LIN {X 0,Y 418.326,Z 381.944,A -85,B 0,C 180,E1 -10142.828,E2 -10142.828} C_VEL
LIN {X 0,Y 420.764,Z 394.079,A -85,B 0,C 180,E1 -10145.581,E2 -10145.581} C_VEL
LIN {X 0,Y 421.234,Z 397.819,A -85,B 0,C 180,E1 -10146.395,E2 -10146.395} C_VEL
LIN {X 0,Y 420.167,Z 413.645,A -85,B 0,C 180,E1 -10149.637,E2 -10149.637} C_VEL
LIN {X 0,Y 419.768,Z 420.199,A -85,B 0,C 180,E1 -10150.945,E2 -10150.945} C_VEL
LIN {X 0,Y 423.831,Z 444.894,A -85,B 0,C 180,E1 -10151.565,E2 -10151.565} C_VEL
LIN {X 0,Y 422.879,Z 528.082,A -85,B 0,C 180,E1 -10152.998,E2 -10152.998} C_VEL
LIN {X 0,Y 422.43,Z 541.332,A -85,B 0,C 180,E1 -10153.415,E2 -10153.415} C_VEL
LIN {X 0,Y 421.773,Z 553.48,A -85,B 0,C 180,E1 -10153.979,E2 -10153.979} C_VEL
LIN {X 0,Y 421.045,Z 565.74,A -85,B 0,C 180,E1 -10154.758,E2 -10154.758} C_VEL
LIN {X 0,Y 420.246,Z 576.923,A -85,B 0,C 180,E1 -10155.68,E2 -10155.68} C_VEL
LIN {X 0,Y 419.549,Z 587.766,A -85,B 0,C 180,E1 -10156.806,E2 -10156.806} C_VEL
LIN {X 0,Y 418.988,Z 596.3,A -85,B 0,C 180,E1 -10157.897,E2 -10157.897} C_VEL
LIN {X 0,Y 418.329,Z 604.171,A -85,B 0,C 180,E1 -10159.105,E2 -10159.105} C_VEL
LIN {X 0,Y 417.793,Z 611.86,A -85,B 0,C 180,E1 -10160.56,E2 -10160.56} C_VEL
LIN {X 0,Y 417.393,Z 618.951,A -85,B 0,C 180,E1 -10162.258,E2 -10162.258} C_VEL
LIN {X 0,Y 417.15,Z 623.713,A -85,B 0,C 180,E1 -10163.728,E2 -10163.728} C_VEL
LIN {X 0,Y 417.114,Z 627.274,A -85,B 0,C 180,E1 -10165.167,E2 -10165.167} C_VEL
LIN {X 0,Y 417,Z 629.132,A -85,B 0,C 180,E1 -10166.134,E2 -10166.134} C_VEL
LIN {X 0,Y 417.018,Z 630.527,A -85,B 0,C 180,E1 -10167.102,E2 -10167.102} C_VEL
LIN {X 0,Y 417.055,Z 631.523,A -85,B 0,C 180,E1 -10168.068,E2 -10168.068} C_VEL
LIN {X 0,Y 416.982,Z 632.345,A -85,B 0,C 180,E1 -10170,E2 -10170} C_VEL
LIN {X 0,Y 417.055,Z 631.522,A -85,B 0,C 180,E1 -10171.931,E2 -10171.931} C_VEL
LIN {X 0,Y 417.018,Z 630.526,A -85,B 0,C 180,E1 -10172.898,E2 -10172.898} C_VEL
LIN {X 0,Y 417,Z 629.129,A -85,B 0,C 180,E1 -10173.865,E2 -10173.865} C_VEL
LIN {X 0,Y 417.137,Z 626.196,A -85,B 0,C 180,E1 -10175.317,E2 -10175.317} C_VEL
LIN {X 0,Y 417.235,Z 622.223,A -85,B 0,C 180,E1 -10176.771,E2 -10176.771} C_VEL
LIN {X 0,Y 417.542,Z 616.116,A -85,B 0,C 180,E1 -10178.469,E2 -10178.469} C_VEL
LIN {X 0,Y 417.955,Z 609.442,A -85,B 0,C 180,E1 -10179.925,E2 -10179.925} C_VEL
LIN {X 0,Y 418.541,Z 601.164,A -85,B 0,C 180,E1 -10181.379,E2 -10181.379} C_VEL
LIN {X 0,Y 419.25,Z 592.68,A -85,B 0,C 180,E1 -10182.587,E2 -10182.587} C_VEL
LIN {X 0,Y 419.898,Z 582.125,A -85,B 0,C 180,E1 -10183.805,E2 -10183.805} C_VEL
LIN {X 0,Y 420.714,Z 570.388,A -85,B 0,C 180,E1 -10184.882,E2 -10184.882} C_VEL
LIN {X 0,Y 421.47,Z 558.517,A -85,B 0,C 180,E1 -10185.722,E2 -10185.722} C_VEL
LIN {X 0,Y 422.196,Z 546.166,A -85,B 0,C 180,E1 -10186.376,E2 -10186.376} C_VEL
LIN {X 0,Y 422.663,Z 533.478,A -85,B 0,C 180,E1 -10186.855,E2 -10186.855} C_VEL
LIN {X 0,Y 423.062,Z 520.188,A -85,B 0,C 180,E1 -10187.149,E2 -10187.149} C_VEL
LIN {X 0,Y 423.713,Z 444.119,A -85,B 0,C 180,E1 -10188.448,E2 -10188.448} C_VEL
LIN {X 0,Y 419.753,Z 419.907,A -85,B 0,C 180,E1 -10189.078,E2 -10189.078} C_VEL
LIN {X 0,Y 421.027,Z 401.735,A -85,B 0,C 180,E1 -10192.787,E2 -10192.787} C_VEL
LIN {X 0,Y 421.181,Z 396.537,A -85,B 0,C 180,E1 -10193.869,E2 -10193.869} C_VEL
LIN {X 0,Y 419.001,Z 385.302,A -85,B 0,C 180,E1 -10196.391,E2 -10196.391} C_VEL
LIN {X 0,Y 418.336,Z 381.878,A -85,B 0,C 180,E1 -10197.208,E2 -10197.208} C_VEL
LIN {X 0,Y 418.247,Z 381.882,A -85,B 0,C 180,E1 -10200.272,E2 -10200.272} C_VEL
LIN {X 0,Y 418.25,Z 381.883,A -85,B 0,C 180,E1 -10203.677,E2 -10203.677} C_VEL
LIN {X 0,Y 418.242,Z 381.888,A -85,B 0,C 180,E1 -10207.224,E2 -10207.224} C_VEL
LIN {X 0,Y 418.253,Z 381.882,A -85,B 0,C 180,E1 -10209.682,E2 -10209.682} C_VEL
LIN {X 0,Y 418.231,Z 381.885,A -85,B 0,C 180,E1 -10212.321,E2 -10212.321} C_VEL
LIN {X 0,Y 418.241,Z 381.888,A -85,B 0,C 180,E1 -10215.109,E2 -10215.109} C_VEL
LIN {X 0,Y 418.244,Z 381.883,A -85,B 0,C 180,E1 -10217.767,E2 -10217.767} C_VEL
LIN {X 0,Y 418.257,Z 381.886,A -85,B 0,C 180,E1 -10220.619,E2 -10220.619} C_VEL
LIN {X 0,Y 418.245,Z 381.883,A -85,B 0,C 180,E1 -10223.976,E2 -10223.976} C_VEL
LIN {X 0,Y 418.259,Z 381.883,A -85,B 0,C 180,E1 -10227.156,E2 -10227.156} C_VEL
LIN {X 0,Y 418.27,Z 381.884,A -85,B 0,C 180,E1 -10230.895,E2 -10230.895} C_VEL
LIN {X 0,Y 418.271,Z 381.881,A -85,B 0,C 180,E1 -10234.096,E2 -10234.096} C_VEL
LIN {X 0,Y 418.24,Z 381.884,A -85,B 0,C 180,E1 -10237.264,E2 -10237.264} C_VEL
LIN {X 0,Y 418.286,Z 381.883,A -85,B 0,C 180,E1 -10240.364,E2 -10240.364} C_VEL
LIN {X 0,Y 418.32,Z 381.873,A -85,B 0,C 180,E1 -10243.405,E2 -10243.405} C_VEL
LIN {X 0,Y 418.358,Z 381.87,A -85,B 0,C 180,E1 -10246.994,E2 -10246.994} C_VEL
LIN {X 0,Y 418.36,Z 381.875,A -85,B 0,C 180,E1 -10250.329,E2 -10250.329} C_VEL
LIN {X 0,Y 418.48,Z 381.853,A -85,B 0,C 180,E1 -10253.249,E2 -10253.249} C_VEL
LIN {X 0,Y 418.341,Z 381.871,A -85,B 0,C 180,E1 -10255.182,E2 -10255.182} C_VEL
LIN {X 0,Y 418.545,Z 381.85,A -85,B 0,C 180,E1 -10258.076,E2 -10258.076} C_VEL
LIN {X 0,Y 418.674,Z 381.834,A -85,B 0,C 180,E1 -10260,E2 -10260} C_VEL
LIN {X 0,Y 418.513,Z 381.85,A -85,B 0,C 180,E1 -10262.888,E2 -10262.888} C_VEL
LIN {X 0,Y 418.497,Z 381.852,A -85,B 0,C 180,E1 -10266.751,E2 -10266.751} C_VEL
LIN {X 0,Y 418.403,Z 381.864,A -85,B 0,C 180,E1 -10268.695,E2 -10268.695} C_VEL
LIN {X 0,Y 418.358,Z 381.87,A -85,B 0,C 180,E1 -10272.614,E2 -10272.614} C_VEL
LIN {X 0,Y 418.305,Z 381.878,A -85,B 0,C 180,E1 -10275.594,E2 -10275.594} C_VEL
LIN {X 0,Y 418.288,Z 381.878,A -85,B 0,C 180,E1 -10278.617,E2 -10278.617} C_VEL
LIN {X 0,Y 418.237,Z 381.888,A -85,B 0,C 180,E1 -10281.696,E2 -10281.696} C_VEL
LIN {X 0,Y 418.286,Z 381.877,A -85,B 0,C 180,E1 -10284.865,E2 -10284.865} C_VEL
LIN {X 0,Y 418.296,Z 381.88,A -85,B 0,C 180,E1 -10288.063,E2 -10288.063} C_VEL
LIN {X 0,Y 418.218,Z 381.889,A -85,B 0,C 180,E1 -10291.396,E2 -10291.396} C_VEL
LIN {X 0,Y 418.268,Z 381.88,A -85,B 0,C 180,E1 -10294.58,E2 -10294.58} C_VEL
LIN {X 0,Y 418.237,Z 381.888,A -85,B 0,C 180,E1 -10297.835,E2 -10297.835} C_VEL
LIN {X 0,Y 418.263,Z 381.881,A -85,B 0,C 180,E1 -10300.943,E2 -10300.943} C_VEL
LIN {X 0,Y 418.219,Z 381.891,A -85,B 0,C 180,E1 -10303.731,E2 -10303.731} C_VEL
LIN {X 0,Y 418.211,Z 381.887,A -85,B 0,C 180,E1 -10306.449,E2 -10306.449} C_VEL
LIN {X 0,Y 418.225,Z 381.888,A -85,B 0,C 180,E1 -10309.13,E2 -10309.13} C_VEL
LIN {X 0,Y 418.236,Z 381.884,A -85,B 0,C 180,E1 -10312.166,E2 -10312.166} C_VEL
LIN {X 0,Y 418.268,Z 381.886,A -85,B 0,C 180,E1 -10315.42,E2 -10315.42} C_VEL
LIN {X 0,Y 418.214,Z 381.887,A -85,B 0,C 180,E1 -10318.604,E2 -10318.604} C_VEL
LIN {X 0,Y 418.294,Z 381.877,A -85,B 0,C 180,E1 -10321.937,E2 -10321.937} C_VEL
LIN {X 0,Y 418.304,Z 381.881,A -85,B 0,C 180,E1 -10325.693,E2 -10325.693} C_VEL
LIN {X 0,Y 418.303,Z 381.998,A -85,B 0,C 180,E1 -10326.121,E2 -10326.121} C_VEL
LIN {X 0,Y 420.404,Z 393.102,A -85,B 0,C 180,E1 -10328.936,E2 -10328.936} C_VEL
LIN {X 0,Y 420.115,Z 399.607,A -85,B 0,C 180,E1 -10330.453,E2 -10330.453} C_VEL
LIN {X 0,Y 419.951,Z 402.004,A -85,B 0,C 180,E1 -10331.004,E2 -10331.004} C_VEL
LIN {X 0,Y 424.021,Z 422.399,A -85,B 0,C 180,E1 -10331.562,E2 -10331.562} C_VEL
LIN {X 0,Y 423.027,Z 509.467,A -85,B 0,C 180,E1 -10333.067,E2 -10333.067} C_VEL
LIN {X 0,Y 422.58,Z 522.544,A -85,B 0,C 180,E1 -10333.484,E2 -10333.484} C_VEL
LIN {X 0,Y 422.003,Z 535.695,A -85,B 0,C 180,E1 -10334.113,E2 -10334.113} C_VEL
LIN {X 0,Y 421.338,Z 547.544,A -85,B 0,C 180,E1 -10334.893,E2 -10334.893} C_VEL
LIN {X 0,Y 420.71,Z 558.93,A -85,B 0,C 180,E1 -10335.861,E2 -10335.861} C_VEL
LIN {X 0,Y 420,Z 569.148,A -85,B 0,C 180,E1 -10336.944,E2 -10336.944} C_VEL
LIN {X 0,Y 419.248,Z 578.338,A -85,B 0,C 180,E1 -10338.15,E2 -10338.15} C_VEL
LIN {X 0,Y 418.538,Z 587.261,A -85,B 0,C 180,E1 -10339.601,E2 -10339.601} C_VEL
LIN {X 0,Y 418.021,Z 594.443,A -85,B 0,C 180,E1 -10341.053,E2 -10341.053} C_VEL
LIN {X 0,Y 417.861,Z 596.308,A -85,B 0,C 180,E1 -10341.496,E2 -10341.496} C_VEL
LIN {X 0,Y 416.976,Z 599.134,A -85,B 0,C 180,E1 -10342.2,E2 -10342.2} C_VEL
LIN {X 0,Y 412.546,Z 604.702,A -85,B 0,C 180,E1 -10343.85,E2 -10343.85} C_VEL
LIN {X 0,Y 410.488,Z 607.256,A -85,B 0,C 180,E1 -10344.856,E2 -10344.856} C_VEL
LIN {X 0,Y 410.102,Z 608.331,A -85,B 0,C 180,E1 -10345.384,E2 -10345.384} C_VEL
LIN {X 0,Y 410.033,Z 611.029,A -85,B 0,C 180,E1 -10347.053,E2 -10347.053} C_VEL
LIN {X 0,Y 410.011,Z 612.026,A -85,B 0,C 180,E1 -10348.036,E2 -10348.036} C_VEL
LIN {X 0,Y 409.907,Z 612.876,A -85,B 0,C 180,E1 -10350,E2 -10350} C_VEL
LIN {X 0,Y 409.939,Z 612.687,A -85,B 0,C 180,E1 -10350.983,E2 -10350.983} C_VEL
LIN {X 0,Y 410.011,Z 612.101,A -85,B 0,C 180,E1 -10351.965,E2 -10351.965} C_VEL
LIN {X 0,Y 410.033,Z 611.134,A -85,B 0,C 180,E1 -10352.948,E2 -10352.948} C_VEL
LIN {X 0,Y 410.02,Z 609.779,A -85,B 0,C 180,E1 -10353.932,E2 -10353.932} C_VEL
LIN {X 0,Y 410.258,Z 606.908,A -85,B 0,C 180,E1 -10355.407,E2 -10355.407} C_VEL
LIN {X 0,Y 410.43,Z 603.021,A -85,B 0,C 180,E1 -10356.885,E2 -10356.885} C_VEL
LIN {X 0,Y 410.747,Z 598.003,A -85,B 0,C 180,E1 -10358.363,E2 -10358.363} C_VEL
LIN {X 0,Y 411.233,Z 591.687,A -85,B 0,C 180,E1 -10359.84,E2 -10359.84} C_VEL
LIN {X 0,Y 411.887,Z 583.778,A -85,B 0,C 180,E1 -10361.316,E2 -10361.316} C_VEL
LIN {X 0,Y 412.532,Z 575.717,A -85,B 0,C 180,E1 -10362.546,E2 -10362.546} C_VEL
LIN {X 0,Y 413.313,Z 565.878,A -85,B 0,C 180,E1 -10363.772,E2 -10363.772} C_VEL
LIN {X 0,Y 414.013,Z 554.816,A -85,B 0,C 180,E1 -10364.878,E2 -10364.878} C_VEL
LIN {X 0,Y 414.727,Z 543.966,A -85,B 0,C 180,E1 -10365.732,E2 -10365.732} C_VEL
LIN {X 0,Y 415.441,Z 531.98,A -85,B 0,C 180,E1 -10366.461,E2 -10366.461} C_VEL
LIN {X 0,Y 415.942,Z 518.813,A -85,B 0,C 180,E1 -10367.041,E2 -10367.041} C_VEL
LIN {X 0,Y 416.334,Z 505.543,A -85,B 0,C 180,E1 -10367.404,E2 -10367.404} C_VEL
LIN {X 0,Y 417.21,Z 422.842,A -85,B 0,C 180,E1 -10368.842,E2 -10368.842} C_VEL
LIN {X 0,Y 413.089,Z 402.156,A -85,B 0,C 180,E1 -10369.42,E2 -10369.42} C_VEL
LIN {X 0,Y 413.501,Z 394.743,A -85,B 0,C 180,E1 -10371.173,E2 -10371.173} C_VEL
LIN {X 0,Y 411.268,Z 382.832,A -85,B 0,C 180,E1 -10374.244,E2 -10374.244} C_VEL
LIN {X 0,Y 411.262,Z 382.758,A -85,B 0,C 180,E1 -10377.478,E2 -10377.478} C_VEL
LIN {X 0,Y 411.193,Z 382.768,A -85,B 0,C 180,E1 -10380.848,E2 -10380.848} C_VEL
LIN {X 0,Y 411.209,Z 382.762,A -85,B 0,C 180,E1 -10384.334,E2 -10384.334} C_VEL
LIN {X 0,Y 411.197,Z 382.761,A -85,B 0,C 180,E1 -10387.974,E2 -10387.974} C_VEL
LIN {X 0,Y 411.167,Z 382.765,A -85,B 0,C 180,E1 -10391.228,E2 -10391.228} C_VEL
LIN {X 0,Y 411.181,Z 382.769,A -85,B 0,C 180,E1 -10394.49,E2 -10394.49} C_VEL
LIN {X 0,Y 411.193,Z 382.764,A -85,B 0,C 180,E1 -10398.196,E2 -10398.196} C_VEL
LIN {X 0,Y 411.228,Z 382.76,A -85,B 0,C 180,E1 -10400.777,E2 -10400.777} C_VEL
LIN {X 0,Y 411.203,Z 382.766,A -85,B 0,C 180,E1 -10404.472,E2 -10404.472} C_VEL
LIN {X 0,Y 411.211,Z 382.76,A -85,B 0,C 180,E1 -10406.873,E2 -10406.873} C_VEL
LIN {X 0,Y 411.243,Z 382.758,A -85,B 0,C 180,E1 -10410.643,E2 -10410.643} C_VEL
LIN {X 0,Y 411.242,Z 382.756,A -85,B 0,C 180,E1 -10413.619,E2 -10413.619} C_VEL
LIN {X 0,Y 411.207,Z 382.76,A -85,B 0,C 180,E1 -10416.853,E2 -10416.853} C_VEL
LIN {X 0,Y 411.269,Z 382.757,A -85,B 0,C 180,E1 -10420.031,E2 -10420.031} C_VEL
LIN {X 0,Y 411.268,Z 382.752,A -85,B 0,C 180,E1 -10423.131,E2 -10423.131} C_VEL
LIN {X 0,Y 411.31,Z 382.746,A -85,B 0,C 180,E1 -10426.896,E2 -10426.896} C_VEL
LIN {X 0,Y 411.297,Z 382.753,A -85,B 0,C 180,E1 -10430.161,E2 -10430.161} C_VEL
LIN {X 0,Y 411.466,Z 382.727,A -85,B 0,C 180,E1 -10433.133,E2 -10433.133} C_VEL
LIN {X 0,Y 411.316,Z 382.746,A -85,B 0,C 180,E1 -10435.099,E2 -10435.099} C_VEL
LIN {X 0,Y 411.517,Z 382.726,A -85,B 0,C 180,E1 -10438.043,E2 -10438.043} C_VEL
LIN {X 0,Y 411.646,Z 382.71,A -85,B 0,C 180,E1 -10440,E2 -10440} C_VEL
LIN {X 0,Y 411.464,Z 382.727,A -85,B 0,C 180,E1 -10442.937,E2 -10442.937} C_VEL
LIN {X 0,Y 411.476,Z 382.731,A -85,B 0,C 180,E1 -10445.882,E2 -10445.882} C_VEL
LIN {X 0,Y 411.327,Z 382.744,A -85,B 0,C 180,E1 -10448.846,E2 -10448.846} C_VEL
LIN {X 0,Y 411.303,Z 382.752,A -85,B 0,C 180,E1 -10451.832,E2 -10451.832} C_VEL
LIN {X 0,Y 411.268,Z 382.752,A -85,B 0,C 180,E1 -10454.852,E2 -10454.852} C_VEL
LIN {X 0,Y 411.257,Z 382.756,A -85,B 0,C 180,E1 -10457.915,E2 -10457.915} C_VEL
LIN {X 0,Y 411.201,Z 382.762,A -85,B 0,C 180,E1 -10461.034,E2 -10461.034} C_VEL
LIN {X 0,Y 411.23,Z 382.757,A -85,B 0,C 180,E1 -10464.215,E2 -10464.215} C_VEL
LIN {X 0,Y 411.263,Z 382.758,A -85,B 0,C 180,E1 -10467.477,E2 -10467.477} C_VEL
LIN {X 0,Y 411.193,Z 382.763,A -85,B 0,C 180,E1 -10470.847,E2 -10470.847} C_VEL
LIN {X 0,Y 411.208,Z 382.759,A -85,B 0,C 180,E1 -10474.333,E2 -10474.333} C_VEL
LIN {X 0,Y 411.197,Z 382.761,A -85,B 0,C 180,E1 -10477.974,E2 -10477.974} C_VEL
LIN {X 0,Y 411.168,Z 382.771,A -85,B 0,C 180,E1 -10481.228,E2 -10481.228} C_VEL
LIN {X 0,Y 411.183,Z 382.763,A -85,B 0,C 180,E1 -10484.49,E2 -10484.49} C_VEL
LIN {X 0,Y 411.181,Z 382.763,A -85,B 0,C 180,E1 -10488.194,E2 -10488.194} C_VEL
LIN {X 0,Y 411.223,Z 382.762,A -85,B 0,C 180,E1 -10490.776,E2 -10490.776} C_VEL
LIN {X 0,Y 411.201,Z 382.762,A -85,B 0,C 180,E1 -10494.471,E2 -10494.471} C_VEL
LIN {X 0,Y 411.21,Z 382.766,A -85,B 0,C 180,E1 -10496.873,E2 -10496.873} C_VEL
LIN {X 0,Y 411.236,Z 382.762,A -85,B 0,C 180,E1 -10500.644,E2 -10500.644} C_VEL
LIN {X 0,Y 411.301,Z 382.856,A -85,B 0,C 180,E1 -10502.56,E2 -10502.56} C_VEL
LIN {X 0,Y 414.008,Z 396.42,A -85,B 0,C 180,E1 -10505.691,E2 -10505.691} C_VEL
LIN {X 0,Y 414.182,Z 401.041,A -85,B 0,C 180,E1 -10506.689,E2 -10506.689} C_VEL
LIN {X 0,Y 412.873,Z 419.278,A -85,B 0,C 180,E1 -10510.485,E2 -10510.485} C_VEL
LIN {X 0,Y 412.845,Z 420.046,A -85,B 0,C 180,E1 -10510.613,E2 -10510.613} C_VEL
LIN {X 0,Y 417.104,Z 446.076,A -85,B 0,C 180,E1 -10511.281,E2 -10511.281} C_VEL
LIN {X 0,Y 416.109,Z 527.927,A -85,B 0,C 180,E1 -10512.713,E2 -10512.713} C_VEL
LIN {X 0,Y 415.634,Z 541.173,A -85,B 0,C 180,E1 -10513.136,E2 -10513.136} C_VEL
LIN {X 0,Y 414.927,Z 553.319,A -85,B 0,C 180,E1 -10513.708,E2 -10513.708} C_VEL
LIN {X 0,Y 414.191,Z 565.577,A -85,B 0,C 180,E1 -10514.499,E2 -10514.499} C_VEL
LIN {X 0,Y 413.33,Z 577.231,A -85,B 0,C 180,E1 -10515.481,E2 -10515.481} C_VEL
LIN {X 0,Y 412.591,Z 587.6,A -85,B 0,C 180,E1 -10516.58,E2 -10516.58} C_VEL
LIN {X 0,Y 412.011,Z 596.134,A -85,B 0,C 180,E1 -10517.688,E2 -10517.688} C_VEL
LIN {X 0,Y 411.34,Z 604.005,A -85,B 0,C 180,E1 -10518.918,E2 -10518.918} C_VEL
LIN {X 0,Y 410.768,Z 611.694,A -85,B 0,C 180,E1 -10520.397,E2 -10520.397} C_VEL
LIN {X 0,Y 410.348,Z 618.785,A -85,B 0,C 180,E1 -10522.125,E2 -10522.125} C_VEL
LIN {X 0,Y 410.048,Z 623.973,A -85,B 0,C 180,E1 -10523.768,E2 -10523.768} C_VEL
LIN {X 0,Y 410.027,Z 627.108,A -85,B 0,C 180,E1 -10525.083,E2 -10525.083} C_VEL
LIN {X 0,Y 409.92,Z 628.966,A -85,B 0,C 180,E1 -10526.067,E2 -10526.067} C_VEL
LIN {X 0,Y 409.965,Z 631.357,A -85,B 0,C 180,E1 -10528.035,E2 -10528.035} C_VEL
LIN {X 0,Y 409.919,Z 631.963,A -85,B 0,C 180,E1 -10529.017,E2 -10529.017} C_VEL
LIN {X 0,Y 409.906,Z 632.178,A -85,B 0,C 180,E1 -10530,E2 -10530} C_VEL
LIN {X 0,Y 409.965,Z 631.355,A -85,B 0,C 180,E1 -10531.965,E2 -10531.965} C_VEL
LIN {X 0,Y 409.92,Z 628.961,A -85,B 0,C 180,E1 -10533.932,E2 -10533.932} C_VEL
LIN {X 0,Y 410.033,Z 626.027,A -85,B 0,C 180,E1 -10535.409,E2 -10535.409} C_VEL
LIN {X 0,Y 410.169,Z 622.055,A -85,B 0,C 180,E1 -10536.889,E2 -10536.889} C_VEL
LIN {X 0,Y 410.49,Z 615.946,A -85,B 0,C 180,E1 -10538.616,E2 -10538.616} C_VEL
LIN {X 0,Y 410.943,Z 609.273,A -85,B 0,C 180,E1 -10540.096,E2 -10540.096} C_VEL
LIN {X 0,Y 411.572,Z 600.994,A -85,B 0,C 180,E1 -10541.574,E2 -10541.574} C_VEL
LIN {X 0,Y 412.286,Z 592.509,A -85,B 0,C 180,E1 -10542.803,E2 -10542.803} C_VEL
LIN {X 0,Y 412.975,Z 581.747,A -85,B 0,C 180,E1 -10544.063,E2 -10544.063} C_VEL
LIN {X 0,Y 413.858,Z 570.218,A -85,B 0,C 180,E1 -10545.135,E2 -10545.135} C_VEL
LIN {X 0,Y 414.644,Z 558.345,A -85,B 0,C 180,E1 -10545.987,E2 -10545.987} C_VEL
LIN {X 0,Y 415.395,Z 545.992,A -85,B 0,C 180,E1 -10546.652,E2 -10546.652} C_VEL
LIN {X 0,Y 415.888,Z 533.301,A -85,B 0,C 180,E1 -10547.138,E2 -10547.138} C_VEL
LIN {X 0,Y 416.286,Z 520.002,A -85,B 0,C 180,E1 -10547.438,E2 -10547.438} C_VEL
LIN {X 0,Y 416.885,Z 444.27,A -85,B 0,C 180,E1 -10548.755,E2 -10548.755} C_VEL
LIN {X 0,Y 412.838,Z 419.847,A -85,B 0,C 180,E1 -10549.387,E2 -10549.387} C_VEL
LIN {X 0,Y 414.212,Z 401.001,A -85,B 0,C 180,E1 -10553.307,E2 -10553.307} C_VEL
LIN {X 0,Y 413.979,Z 396.375,A -85,B 0,C 180,E1 -10554.311,E2 -10554.311} C_VEL
LIN {X 0,Y 411.302,Z 382.808,A -85,B 0,C 180,E1 -10557.441,E2 -10557.441} C_VEL
LIN {X 0,Y 411.191,Z 382.765,A -85,B 0,C 180,E1 -10560.847,E2 -10560.847} C_VEL
LIN {X 0,Y 411.208,Z 382.76,A -85,B 0,C 180,E1 -10564.333,E2 -10564.333} C_VEL
LIN {X 0,Y 411.197,Z 382.76,A -85,B 0,C 180,E1 -10567.973,E2 -10567.973} C_VEL
LIN {X 0,Y 411.183,Z 382.764,A -85,B 0,C 180,E1 -10570.504,E2 -10570.504} C_VEL
LIN {X 0,Y 411.175,Z 382.768,A -85,B 0,C 180,E1 -10573.133,E2 -10573.133} C_VEL
LIN {X 0,Y 411.174,Z 382.763,A -85,B 0,C 180,E1 -10575.88,E2 -10575.88} C_VEL
LIN {X 0,Y 411.167,Z 382.771,A -85,B 0,C 180,E1 -10578.771,E2 -10578.771} C_VEL
LIN {X 0,Y 411.208,Z 382.759,A -85,B 0,C 180,E1 -10581.831,E2 -10581.831} C_VEL
LIN {X 0,Y 411.212,Z 382.762,A -85,B 0,C 180,E1 -10585.121,E2 -10585.121} C_VEL
LIN {X 0,Y 411.168,Z 382.765,A -85,B 0,C 180,E1 -10588.003,E2 -10588.003} C_VEL
LIN {X 0,Y 411.22,Z 382.758,A -85,B 0,C 180,E1 -10591.41,E2 -10591.41} C_VEL
LIN {X 0,Y 411.239,Z 382.755,A -85,B 0,C 180,E1 -10593.619,E2 -10593.619} C_VEL
LIN {X 0,Y 411.204,Z 382.763,A -85,B 0,C 180,E1 -10596.852,E2 -10596.852} C_VEL
LIN {X 0,Y 411.217,Z 382.76,A -85,B 0,C 180,E1 -10600.05,E2 -10600.05} C_VEL
LIN {X 0,Y 411.265,Z 382.753,A -85,B 0,C 180,E1 -10603.131,E2 -10603.131} C_VEL
LIN {X 0,Y 411.316,Z 382.748,A -85,B 0,C 180,E1 -10606.891,E2 -10606.891} C_VEL
LIN {X 0,Y 411.309,Z 382.751,A -85,B 0,C 180,E1 -10610.162,E2 -10610.162} C_VEL
LIN {X 0,Y 411.444,Z 382.73,A -85,B 0,C 180,E1 -10613.133,E2 -10613.133} C_VEL
LIN {X 0,Y 411.312,Z 382.746,A -85,B 0,C 180,E1 -10615.099,E2 -10615.099} C_VEL
LIN {X 0,Y 411.514,Z 382.726,A -85,B 0,C 180,E1 -10618.043,E2 -10618.043} C_VEL
LIN {X 0,Y 411.643,Z 382.71,A -85,B 0,C 180,E1 -10620,E2 -10620} C_VEL
LIN {X 0,Y 411.469,Z 382.727,A -85,B 0,C 180,E1 -10622.937,E2 -10622.937} C_VEL
LIN {X 0,Y 411.464,Z 382.728,A -85,B 0,C 180,E1 -10626.867,E2 -10626.867} C_VEL
LIN {X 0,Y 411.295,Z 382.753,A -85,B 0,C 180,E1 -10629.839,E2 -10629.839} C_VEL
LIN {X 0,Y 411.308,Z 382.747,A -85,B 0,C 180,E1 -10633.104,E2 -10633.104} C_VEL
LIN {X 0,Y 411.265,Z 382.752,A -85,B 0,C 180,E1 -10636.869,E2 -10636.869} C_VEL
LIN {X 0,Y 411.257,Z 382.759,A -85,B 0,C 180,E1 -10639.986,E2 -10639.986} C_VEL
LIN {X 0,Y 411.206,Z 382.76,A -85,B 0,C 180,E1 -10643.148,E2 -10643.148} C_VEL
LIN {X 0,Y 411.241,Z 382.756,A -85,B 0,C 180,E1 -10646.381,E2 -10646.381} C_VEL
LIN {X 0,Y 411.211,Z 382.766,A -85,B 0,C 180,E1 -10649.712,E2 -10649.712} C_VEL
LIN {X 0,Y 411.208,Z 382.761,A -85,B 0,C 180,E1 -10653.156,E2 -10653.156} C_VEL
LIN {X 0,Y 411.198,Z 382.76,A -85,B 0,C 180,E1 -10656.553,E2 -10656.553} C_VEL
LIN {X 0,Y 411.221,Z 382.763,A -85,B 0,C 180,E1 -10659.729,E2 -10659.729} C_VEL
LIN {X 0,Y 411.18,Z 382.765,A -85,B 0,C 180,E1 -10663.133,E2 -10663.133} C_VEL
LIN {X 0,Y 411.17,Z 382.767,A -85,B 0,C 180,E1 -10665.881,E2 -10665.881} C_VEL
LIN {X 0,Y 411.165,Z 382.765,A -85,B 0,C 180,E1 -10668.772,E2 -10668.772} C_VEL
LIN {X 0,Y 411.201,Z 382.761,A -85,B 0,C 180,E1 -10672.027,E2 -10672.027} C_VEL
LIN {X 0,Y 411.209,Z 382.762,A -85,B 0,C 180,E1 -10675.667,E2 -10675.667} C_VEL
LIN {X 0,Y 411.192,Z 382.767,A -85,B 0,C 180,E1 -10679.153,E2 -10679.153} C_VEL
LIN {X 0,Y 411.261,Z 382.753,A -85,B 0,C 180,E1 -10682.523,E2 -10682.523} C_VEL
LIN {X 0,Y 411.3,Z 382.817,A -85,B 0,C 180,E1 -10685.856,E2 -10685.856} C_VEL
LIN {X 0,Y 413.452,Z 394.335,A -85,B 0,C 180,E1 -10688.825,E2 -10688.825} C_VEL
LIN {X 0,Y 413.245,Z 399.77,A -85,B 0,C 180,E1 -10690.115,E2 -10690.115} C_VEL
LIN {X 0,Y 413.08,Z 402.168,A -85,B 0,C 180,E1 -10690.676,E2 -10690.676} C_VEL
LIN {X 0,Y 417.325,Z 423.697,A -85,B 0,C 180,E1 -10691.275,E2 -10691.275} C_VEL
LIN {X 0,Y 416.256,Z 509.651,A -85,B 0,C 180,E1 -10692.783,E2 -10692.783} C_VEL
LIN {X 0,Y 415.747,Z 523.483,A -85,B 0,C 180,E1 -10693.236,E2 -10693.236} C_VEL
LIN {X 0,Y 415.17,Z 535.871,A -85,B 0,C 180,E1 -10693.844,E2 -10693.844} C_VEL
LIN {X 0,Y 414.492,Z 547.717,A -85,B 0,C 180,E1 -10694.637,E2 -10694.637} C_VEL
LIN {X 0,Y 413.824,Z 559.102,A -85,B 0,C 180,E1 -10695.621,E2 -10695.621} C_VEL
LIN {X 0,Y 413.08,Z 569.319,A -85,B 0,C 180,E1 -10696.722,E2 -10696.722} C_VEL
LIN {X 0,Y 412.309,Z 578.508,A -85,B 0,C 180,E1 -10697.948,E2 -10697.948} C_VEL
LIN {X 0,Y 411.558,Z 587.43,A -85,B 0,C 180,E1 -10699.422,E2 -10699.422} C_VEL
LIN {X 0,Y 410.993,Z 594.612,A -85,B 0,C 180,E1 -10700.899,E2 -10700.899} C_VEL
LIN {X 0,Y 410.612,Z 599.456,A -85,B 0,C 180,E1 -10702.13,E2 -10702.13} C_VEL
LIN {X 0,Y 410.33,Z 604.475,A -85,B 0,C 180,E1 -10703.717,E2 -10703.717} C_VEL
LIN {X 0,Y 410.155,Z 607.765,A -85,B 0,C 180,E1 -10705.085,E2 -10705.085} C_VEL
LIN {X 0,Y 410.102,Z 608.331,A -85,B 0,C 180,E1 -10705.384,E2 -10705.384} C_VEL
LIN {X 0,Y 409.34,Z 609.832,A -85,B 0,C 180,E1 -10706.18,E2 -10706.18} C_VEL
LIN {X 0,Y 406.396,Z 611.633,A -85,B 0,C 180,E1 -10707.487,E2 -10707.487} C_VEL
LIN {X 0,Y 403.958,Z 612.567,A -85,B 0,C 180,E1 -10708.553,E2 -10708.553} C_VEL
LIN {X 0,Y 402.916,Z 612.943,A -85,B 0,C 180,E1 -10709.383,E2 -10709.383} C_VEL
LIN {X 0,Y 402.831,Z 612.963,A -85,B 0,C 180,E1 -10709.664,E2 -10709.664} C_VEL
LIN {X 0,Y 402.867,Z 612.853,A -85,B 0,C 180,E1 -10711,E2 -10711} C_VEL
LIN {X 0,Y 402.925,Z 612.267,A -85,B 0,C 180,E1 -10711.999,E2 -10711.999} C_VEL
LIN {X 0,Y 402.934,Z 611.301,A -85,B 0,C 180,E1 -10713,E2 -10713} C_VEL
LIN {X 0,Y 402.94,Z 609.945,A -85,B 0,C 180,E1 -10714.001,E2 -10714.001} C_VEL
LIN {X 0,Y 403.183,Z 607.075,A -85,B 0,C 180,E1 -10715.502,E2 -10715.502} C_VEL
LIN {X 0,Y 403.365,Z 603.187,A -85,B 0,C 180,E1 -10717.006,E2 -10717.006} C_VEL
LIN {X 0,Y 403.7,Z 598.169,A -85,B 0,C 180,E1 -10718.51,E2 -10718.51} C_VEL
LIN {X 0,Y 404.213,Z 591.852,A -85,B 0,C 180,E1 -10720.013,E2 -10720.013} C_VEL
LIN {X 0,Y 404.891,Z 583.943,A -85,B 0,C 180,E1 -10721.515,E2 -10721.515} C_VEL
LIN {X 0,Y 405.61,Z 575.881,A -85,B 0,C 180,E1 -10722.763,E2 -10722.763} C_VEL
LIN {X 0,Y 406.411,Z 566.042,A -85,B 0,C 180,E1 -10724.011,E2 -10724.011} C_VEL
LIN {X 0,Y 407.159,Z 554.978,A -85,B 0,C 180,E1 -10725.134,E2 -10725.134} C_VEL
LIN {X 0,Y 407.9,Z 544.126,A -85,B 0,C 180,E1 -10726.003,E2 -10726.003} C_VEL
LIN {X 0,Y 408.651,Z 532.138,A -85,B 0,C 180,E1 -10726.743,E2 -10726.743} C_VEL
LIN {X 0,Y 409.171,Z 518.966,A -85,B 0,C 180,E1 -10727.332,E2 -10727.332} C_VEL
LIN {X 0,Y 409.568,Z 505.688,A -85,B 0,C 180,E1 -10727.701,E2 -10727.701} C_VEL
LIN {X 0,Y 410.543,Z 424.086,A -85,B 0,C 180,E1 -10729.14,E2 -10729.14} C_VEL
LIN {X 0,Y 406.205,Z 402.235,A -85,B 0,C 180,E1 -10729.783,E2 -10729.783} C_VEL
LIN {X 0,Y 406.563,Z 395.983,A -85,B 0,C 180,E1 -10731.286,E2 -10731.286} C_VEL
LIN {X 0,Y 404.225,Z 383.642,A -85,B 0,C 180,E1 -10734.526,E2 -10734.526} C_VEL
LIN {X 0,Y 404.199,Z 383.634,A -85,B 0,C 180,E1 -10738,E2 -10738} C_VEL
LIN {X 0,Y 404.143,Z 383.64,A -85,B 0,C 180,E1 -10741.558,E2 -10741.558} C_VEL
LIN {X 0,Y 404.188,Z 383.637,A -85,B 0,C 180,E1 -10745.016,E2 -10745.016} C_VEL
LIN {X 0,Y 404.156,Z 383.644,A -85,B 0,C 180,E1 -10748.757,E2 -10748.757} C_VEL
LIN {X 0,Y 404.126,Z 383.641,A -85,B 0,C 180,E1 -10751.6,E2 -10751.6} C_VEL
LIN {X 0,Y 404.15,Z 383.645,A -85,B 0,C 180,E1 -10754.522,E2 -10754.522} C_VEL
LIN {X 0,Y 404.144,Z 383.639,A -85,B 0,C 180,E1 -10757.296,E2 -10757.296} C_VEL
LIN {X 0,Y 404.173,Z 383.637,A -85,B 0,C 180,E1 -10759.956,E2 -10759.956} C_VEL
LIN {X 0,Y 404.144,Z 383.64,A -85,B 0,C 180,E1 -10763.125,E2 -10763.125} C_VEL
LIN {X 0,Y 404.149,Z 383.643,A -85,B 0,C 180,E1 -10766.188,E2 -10766.188} C_VEL
LIN {X 0,Y 404.157,Z 383.639,A -85,B 0,C 180,E1 -10769.716,E2 -10769.716} C_VEL
LIN {X 0,Y 404.199,Z 383.632,A -85,B 0,C 180,E1 -10773.123,E2 -10773.123} C_VEL
LIN {X 0,Y 404.181,Z 383.635,A -85,B 0,C 180,E1 -10775.334,E2 -10775.334} C_VEL
LIN {X 0,Y 404.168,Z 383.639,A -85,B 0,C 180,E1 -10778.582,E2 -10778.582} C_VEL
LIN {X 0,Y 404.219,Z 383.633,A -85,B 0,C 180,E1 -10781.762,E2 -10781.762} C_VEL
LIN {X 0,Y 404.212,Z 383.631,A -85,B 0,C 180,E1 -10784.882,E2 -10784.882} C_VEL
LIN {X 0,Y 404.261,Z 383.631,A -85,B 0,C 180,E1 -10787.959,E2 -10787.959} C_VEL
LIN {X 0,Y 404.438,Z 383.608,A -85,B 0,C 180,E1 -10792.1,E2 -10792.1} C_VEL
LIN {X 0,Y 404.429,Z 383.61,A -85,B 0,C 180,E1 -10794.015,E2 -10794.015} C_VEL
LIN {X 0,Y 404.486,Z 383.602,A -85,B 0,C 180,E1 -10798.008,E2 -10798.008} C_VEL
LIN {X 0,Y 404.615,Z 383.586,A -85,B 0,C 180,E1 -10800,E2 -10800} C_VEL
LIN {X 0,Y 404.422,Z 383.605,A -85,B 0,C 180,E1 -10802.988,E2 -10802.988} C_VEL
LIN {X 0,Y 404.424,Z 383.608,A -85,B 0,C 180,E1 -10805.985,E2 -10805.985} C_VEL
LIN {X 0,Y 404.275,Z 383.623,A -85,B 0,C 180,E1 -10809.001,E2 -10809.001} C_VEL
LIN {X 0,Y 404.274,Z 383.625,A -85,B 0,C 180,E1 -10812.041,E2 -10812.041} C_VEL
LIN {X 0,Y 404.213,Z 383.633,A -85,B 0,C 180,E1 -10815.118,E2 -10815.118} C_VEL
LIN {X 0,Y 404.215,Z 383.631,A -85,B 0,C 180,E1 -10818.238,E2 -10818.238} C_VEL
LIN {X 0,Y 404.165,Z 383.643,A -85,B 0,C 180,E1 -10821.418,E2 -10821.418} C_VEL
LIN {X 0,Y 404.181,Z 383.635,A -85,B 0,C 180,E1 -10824.665,E2 -10824.665} C_VEL
LIN {X 0,Y 404.199,Z 383.633,A -85,B 0,C 180,E1 -10827.999,E2 -10827.999} C_VEL
LIN {X 0,Y 404.143,Z 383.643,A -85,B 0,C 180,E1 -10831.558,E2 -10831.558} C_VEL
LIN {X 0,Y 404.187,Z 383.638,A -85,B 0,C 180,E1 -10835.016,E2 -10835.016} C_VEL
LIN {X 0,Y 404.156,Z 383.64,A -85,B 0,C 180,E1 -10838.757,E2 -10838.757} C_VEL
LIN {X 0,Y 404.127,Z 383.643,A -85,B 0,C 180,E1 -10841.6,E2 -10841.6} C_VEL
LIN {X 0,Y 404.152,Z 383.639,A -85,B 0,C 180,E1 -10844.522,E2 -10844.522} C_VEL
LIN {X 0,Y 404.14,Z 383.644,A -85,B 0,C 180,E1 -10847.295,E2 -10847.295} C_VEL
LIN {X 0,Y 404.172,Z 383.636,A -85,B 0,C 180,E1 -10849.955,E2 -10849.955} C_VEL
LIN {X 0,Y 404.14,Z 383.645,A -85,B 0,C 180,E1 -10853.125,E2 -10853.125} C_VEL
LIN {X 0,Y 404.148,Z 383.639,A -85,B 0,C 180,E1 -10856.188,E2 -10856.188} C_VEL
LIN {X 0,Y 404.149,Z 383.643,A -85,B 0,C 180,E1 -10859.715,E2 -10859.715} C_VEL
LIN {X 0,Y 404.241,Z 383.771,A -85,B 0,C 180,E1 -10862.28,E2 -10862.28} C_VEL
LIN {X 0,Y 407.028,Z 397.507,A -85,B 0,C 180,E1 -10865.518,E2 -10865.518} C_VEL
LIN {X 0,Y 407.34,Z 400.903,A -85,B 0,C 180,E1 -10866.278,E2 -10866.278} C_VEL
LIN {X 0,Y 406.109,Z 417.273,A -85,B 0,C 180,E1 -10869.75,E2 -10869.75} C_VEL
LIN {X 0,Y 405.972,Z 419.894,A -85,B 0,C 180,E1 -10870.271,E2 -10870.271} C_VEL
LIN {X 0,Y 410.373,Z 446.646,A -85,B 0,C 180,E1 -10870.975,E2 -10870.975} C_VEL
LIN {X 0,Y 409.34,Z 527.772,A -85,B 0,C 180,E1 -10872.418,E2 -10872.418} C_VEL
LIN {X 0,Y 408.845,Z 541.014,A -85,B 0,C 180,E1 -10872.847,E2 -10872.847} C_VEL
LIN {X 0,Y 408.129,Z 553.158,A -85,B 0,C 180,E1 -10873.428,E2 -10873.428} C_VEL
LIN {X 0,Y 407.323,Z 565.413,A -85,B 0,C 180,E1 -10874.231,E2 -10874.231} C_VEL
LIN {X 0,Y 406.426,Z 577.259,A -85,B 0,C 180,E1 -10875.248,E2 -10875.248} C_VEL
LIN {X 0,Y 405.577,Z 588.478,A -85,B 0,C 180,E1 -10876.471,E2 -10876.471} C_VEL
LIN {X 0,Y 404.897,Z 597.645,A -85,B 0,C 180,E1 -10877.723,E2 -10877.723} C_VEL
LIN {X 0,Y 404.1,Z 606.575,A -85,B 0,C 180,E1 -10879.224,E2 -10879.224} C_VEL
LIN {X 0,Y 403.562,Z 613.764,A -85,B 0,C 180,E1 -10880.73,E2 -10880.73} C_VEL
LIN {X 0,Y 403.292,Z 618.618,A -85,B 0,C 180,E1 -10881.986,E2 -10881.986} C_VEL
LIN {X 0,Y 402.958,Z 624.153,A -85,B 0,C 180,E1 -10883.795,E2 -10883.795} C_VEL
LIN {X 0,Y 402.94,Z 626.941,A -85,B 0,C 180,E1 -10884.997,E2 -10884.997} C_VEL
LIN {X 0,Y 402.842,Z 628.799,A -85,B 0,C 180,E1 -10885.998,E2 -10885.998} C_VEL
LIN {X 0,Y 402.862,Z 631.19,A -85,B 0,C 180,E1 -10888,E2 -10888} C_VEL
LIN {X 0,Y 402.847,Z 631.797,A -85,B 0,C 180,E1 -10889,E2 -10889} C_VEL
LIN {X 0,Y 402.832,Z 632.011,A -85,B 0,C 180,E1 -10890,E2 -10890} C_VEL
LIN {X 0,Y 402.847,Z 631.795,A -85,B 0,C 180,E1 -10890.999,E2 -10890.999} C_VEL
LIN {X 0,Y 402.862,Z 631.187,A -85,B 0,C 180,E1 -10891.999,E2 -10891.999} C_VEL
LIN {X 0,Y 402.842,Z 628.794,A -85,B 0,C 180,E1 -10894.001,E2 -10894.001} C_VEL
LIN {X 0,Y 402.934,Z 625.859,A -85,B 0,C 180,E1 -10895.505,E2 -10895.505} C_VEL
LIN {X 0,Y 403.083,Z 621.886,A -85,B 0,C 180,E1 -10897.01,E2 -10897.01} C_VEL
LIN {X 0,Y 403.428,Z 615.777,A -85,B 0,C 180,E1 -10898.768,E2 -10898.768} C_VEL
LIN {X 0,Y 403.936,Z 609.104,A -85,B 0,C 180,E1 -10900.273,E2 -10900.273} C_VEL
LIN {X 0,Y 404.602,Z 600.825,A -85,B 0,C 180,E1 -10901.777,E2 -10901.777} C_VEL
LIN {X 0,Y 405.331,Z 592.339,A -85,B 0,C 180,E1 -10903.027,E2 -10903.027} C_VEL
LIN {X 0,Y 406.02,Z 582.348,A -85,B 0,C 180,E1 -10904.226,E2 -10904.226} C_VEL
LIN {X 0,Y 406.863,Z 571.475,A -85,B 0,C 180,E1 -10905.273,E2 -10905.273} C_VEL
LIN {X 0,Y 407.668,Z 560.099,A -85,B 0,C 180,E1 -10906.14,E2 -10906.14} C_VEL
LIN {X 0,Y 408.398,Z 548.419,A -85,B 0,C 180,E1 -10906.817,E2 -10906.817} C_VEL
LIN {X 0,Y 409.043,Z 534.956,A -85,B 0,C 180,E1 -10907.369,E2 -10907.369} C_VEL
LIN {X 0,Y 409.499,Z 521.604,A -85,B 0,C 180,E1 -10907.704,E2 -10907.704} C_VEL
LIN {X 0,Y 410.224,Z 445.447,A -85,B 0,C 180,E1 -10909.046,E2 -10909.046} C_VEL
LIN {X 0,Y 405.934,Z 419.68,A -85,B 0,C 180,E1 -10909.731,E2 -10909.731} C_VEL
LIN {X 0,Y 407.252,Z 402.427,A -85,B 0,C 180,E1 -10913.385,E2 -10913.385} C_VEL
LIN {X 0,Y 407.286,Z 399.175,A -85,B 0,C 180,E1 -10914.091,E2 -10914.091} C_VEL
LIN {X 0,Y 405.029,Z 387.491,A -85,B 0,C 180,E1 -10916.817,E2 -10916.817} C_VEL
LIN {X 0,Y 404.211,Z 383.637,A -85,B 0,C 180,E1 -10917.791,E2 -10917.791} C_VEL
LIN {X 0,Y 404.144,Z 383.642,A -85,B 0,C 180,E1 -10921.446,E2 -10921.446} C_VEL
LIN {X 0,Y 404.186,Z 383.64,A -85,B 0,C 180,E1 -10925.016,E2 -10925.016} C_VEL
LIN {X 0,Y 404.157,Z 383.641,A -85,B 0,C 180,E1 -10928.757,E2 -10928.757} C_VEL
LIN {X 0,Y 404.125,Z 383.642,A -85,B 0,C 180,E1 -10931.6,E2 -10931.6} C_VEL
LIN {X 0,Y 404.148,Z 383.641,A -85,B 0,C 180,E1 -10934.522,E2 -10934.522} C_VEL
LIN {X 0,Y 404.141,Z 383.642,A -85,B 0,C 180,E1 -10937.296,E2 -10937.296} C_VEL
LIN {X 0,Y 404.17,Z 383.636,A -85,B 0,C 180,E1 -10939.955,E2 -10939.955} C_VEL
LIN {X 0,Y 404.138,Z 383.643,A -85,B 0,C 180,E1 -10943.125,E2 -10943.125} C_VEL
LIN {X 0,Y 404.146,Z 383.64,A -85,B 0,C 180,E1 -10946.188,E2 -10946.188} C_VEL
LIN {X 0,Y 404.147,Z 383.639,A -85,B 0,C 180,E1 -10949.715,E2 -10949.715} C_VEL
LIN {X 0,Y 404.197,Z 383.634,A -85,B 0,C 180,E1 -10953.123,E2 -10953.123} C_VEL
LIN {X 0,Y 404.178,Z 383.635,A -85,B 0,C 180,E1 -10955.334,E2 -10955.334} C_VEL
LIN {X 0,Y 404.162,Z 383.644,A -85,B 0,C 180,E1 -10958.582,E2 -10958.582} C_VEL
LIN {X 0,Y 404.212,Z 383.631,A -85,B 0,C 180,E1 -10961.762,E2 -10961.762} C_VEL
LIN {X 0,Y 404.211,Z 383.633,A -85,B 0,C 180,E1 -10964.882,E2 -10964.882} C_VEL
LIN {X 0,Y 404.272,Z 383.625,A -85,B 0,C 180,E1 -10967.959,E2 -10967.959} C_VEL
LIN {X 0,Y 404.273,Z 383.624,A -85,B 0,C 180,E1 -10970.999,E2 -10970.999} C_VEL
LIN {X 0,Y 404.419,Z 383.608,A -85,B 0,C 180,E1 -10974.015,E2 -10974.015} C_VEL
LIN {X 0,Y 404.483,Z 383.601,A -85,B 0,C 180,E1 -10978.009,E2 -10978.009} C_VEL
LIN {X 0,Y 404.612,Z 383.585,A -85,B 0,C 180,E1 -10980,E2 -10980} C_VEL
LIN {X 0,Y 404.426,Z 383.604,A -85,B 0,C 180,E1 -10982.988,E2 -10982.988} C_VEL
LIN {X 0,Y 404.415,Z 383.605,A -85,B 0,C 180,E1 -10986.987,E2 -10986.987} C_VEL
LIN {X 0,Y 404.26,Z 383.631,A -85,B 0,C 180,E1 -10990.012,E2 -10990.012} C_VEL
LIN {X 0,Y 404.269,Z 383.624,A -85,B 0,C 180,E1 -10993.211,E2 -10993.211} C_VEL
LIN {X 0,Y 404.218,Z 383.63,A -85,B 0,C 180,E1 -10997.007,E2 -10997.007} C_VEL
LIN {X 0,Y 404.2,Z 383.634,A -85,B 0,C 180,E1 -11000.35,E2 -11000.35} C_VEL
LIN {X 0,Y 404.172,Z 383.639,A -85,B 0,C 180,E1 -11003.574,E2 -11003.574} C_VEL
LIN {X 0,Y 404.186,Z 383.641,A -85,B 0,C 180,E1 -11005.766,E2 -11005.766} C_VEL
LIN {X 0,Y 404.199,Z 383.637,A -85,B 0,C 180,E1 -11008,E2 -11008} C_VEL
LIN {X 0,Y 404.144,Z 383.644,A -85,B 0,C 180,E1 -11011.559,E2 -11011.559} C_VEL
LIN {X 0,Y 404.188,Z 383.634,A -85,B 0,C 180,E1 -11015.016,E2 -11015.016} C_VEL
LIN {X 0,Y 404.161,Z 383.637,A -85,B 0,C 180,E1 -11018.756,E2 -11018.756} C_VEL
LIN {X 0,Y 404.144,Z 383.646,A -85,B 0,C 180,E1 -11021.603,E2 -11021.603} C_VEL
LIN {X 0,Y 404.151,Z 383.638,A -85,B 0,C 180,E1 -11024.523,E2 -11024.523} C_VEL
LIN {X 0,Y 404.138,Z 383.645,A -85,B 0,C 180,E1 -11027.296,E2 -11027.296} C_VEL
LIN {X 0,Y 404.171,Z 383.637,A -85,B 0,C 180,E1 -11029.956,E2 -11029.956} C_VEL
LIN {X 0,Y 404.142,Z 383.643,A -85,B 0,C 180,E1 -11033.124,E2 -11033.124} C_VEL
LIN {X 0,Y 404.147,Z 383.639,A -85,B 0,C 180,E1 -11036.188,E2 -11036.188} C_VEL
LIN {X 0,Y 404.148,Z 383.641,A -85,B 0,C 180,E1 -11039.715,E2 -11039.715} C_VEL
LIN {X 0,Y 404.198,Z 383.638,A -85,B 0,C 180,E1 -11043.123,E2 -11043.123} C_VEL
LIN {X 0,Y 404.26,Z 383.772,A -85,B 0,C 180,E1 -11045.614,E2 -11045.614} C_VEL
LIN {X 0,Y 406.478,Z 395.575,A -85,B 0,C 180,E1 -11048.71,E2 -11048.71} C_VEL
LIN {X 0,Y 406.189,Z 402.293,A -85,B 0,C 180,E1 -11050.324,E2 -11050.324} C_VEL
LIN {X 0,Y 410.54,Z 424.161,A -85,B 0,C 180,E1 -11050.959,E2 -11050.959} C_VEL
LIN {X 0,Y 409.503,Z 509.834,A -85,B 0,C 180,E1 -11052.49,E2 -11052.49} C_VEL
LIN {X 0,Y 408.968,Z 523.661,A -85,B 0,C 180,E1 -11052.95,E2 -11052.95} C_VEL
LIN {X 0,Y 408.368,Z 536.045,A -85,B 0,C 180,E1 -11053.567,E2 -11053.567} C_VEL
LIN {X 0,Y 407.662,Z 547.89,A -85,B 0,C 180,E1 -11054.373,E2 -11054.373} C_VEL
LIN {X 0,Y 406.985,Z 558.009,A -85,B 0,C 180,E1 -11055.248,E2 -11055.248} C_VEL
LIN {X 0,Y 406.234,Z 568.43,A -85,B 0,C 180,E1 -11056.366,E2 -11056.366} C_VEL
LIN {X 0,Y 405.506,Z 576.983,A -85,B 0,C 180,E1 -11057.488,E2 -11057.488} C_VEL
LIN {X 0,Y 404.846,Z 584.859,A -85,B 0,C 180,E1 -11058.738,E2 -11058.738} C_VEL
LIN {X 0,Y 404.18,Z 592.56,A -85,B 0,C 180,E1 -11060.239,E2 -11060.239} C_VEL
LIN {X 0,Y 403.586,Z 599.625,A -85,B 0,C 180,E1 -11061.992,E2 -11061.992} C_VEL
LIN {X 0,Y 403.309,Z 603.928,A -85,B 0,C 180,E1 -11063.353,E2 -11063.353} C_VEL
LIN {X 0,Y 403.1,Z 607.933,A -85,B 0,C 180,E1 -11064.999,E2 -11064.999} C_VEL
LIN {X 0,Y 402.943,Z 609.796,A -85,B 0,C 180,E1 -11066,E2 -11066} C_VEL
LIN {X 0,Y 402.935,Z 611.197,A -85,B 0,C 180,E1 -11067.001,E2 -11067.001} C_VEL
LIN {X 0,Y 402.925,Z 612.193,A -85,B 0,C 180,E1 -11068.001,E2 -11068.001} C_VEL
LIN {X 0,Y 402.831,Z 612.963,A -85,B 0,C 180,E1 -11069.664,E2 -11069.664} C_VEL
LIN {X 0,Y 402.157,Z 613.017,A -85,B 0,C 180,E1 -11070.498,E2 -11070.498} C_VEL
LIN {X 0,Y 399.296,Z 612.483,A -85,B 0,C 180,E1 -11071.853,E2 -11071.853} C_VEL
LIN {X 0,Y 396.906,Z 611.556,A -85,B 0,C 180,E1 -11072.942,E2 -11072.942} C_VEL
LIN {X 0,Y 395.921,Z 610.526,A -85,B 0,C 180,E1 -11073.778,E2 -11073.778} C_VEL
LIN {X 0,Y 395.863,Z 610.128,A -85,B 0,C 180,E1 -11074.06,E2 -11074.06} C_VEL
LIN {X 0,Y 396.113,Z 607.241,A -85,B 0,C 180,E1 -11075.6,E2 -11075.6} C_VEL
LIN {X 0,Y 396.308,Z 603.353,A -85,B 0,C 180,E1 -11077.131,E2 -11077.131} C_VEL
LIN {X 0,Y 396.666,Z 598.335,A -85,B 0,C 180,E1 -11078.662,E2 -11078.662} C_VEL
LIN {X 0,Y 397.22,Z 592.017,A -85,B 0,C 180,E1 -11080.191,E2 -11080.191} C_VEL
LIN {X 0,Y 397.911,Z 584.109,A -85,B 0,C 180,E1 -11081.719,E2 -11081.719} C_VEL
LIN {X 0,Y 398.848,Z 574.268,A -85,B 0,C 180,E1 -11083.243,E2 -11083.243} C_VEL
LIN {X 0,Y 399.687,Z 564.726,A -85,B 0,C 180,E1 -11084.424,E2 -11084.424} C_VEL
LIN {X 0,Y 400.403,Z 553.717,A -85,B 0,C 180,E1 -11085.526,E2 -11085.526} C_VEL
LIN {X 0,Y 401.251,Z 542.524,A -85,B 0,C 180,E1 -11086.406,E2 -11086.406} C_VEL
LIN {X 0,Y 401.932,Z 531.167,A -85,B 0,C 180,E1 -11087.096,E2 -11087.096} C_VEL
LIN {X 0,Y 402.471,Z 518.205,A -85,B 0,C 180,E1 -11087.663,E2 -11087.663} C_VEL
LIN {X 0,Y 402.861,Z 504.328,A -85,B 0,C 180,E1 -11088.039,E2 -11088.039} C_VEL
LIN {X 0,Y 403.855,Z 425.441,A -85,B 0,C 180,E1 -11089.447,E2 -11089.447} C_VEL
LIN {X 0,Y 399.347,Z 402.391,A -85,B 0,C 180,E1 -11090.138,E2 -11090.138} C_VEL
LIN {X 0,Y 399.628,Z 397.882,A -85,B 0,C 180,E1 -11091.238,E2 -11091.238} C_VEL
LIN {X 0,Y 397.776,Z 387.53,A -85,B 0,C 180,E1 -11093.977,E2 -11093.977} C_VEL
LIN {X 0,Y 397.167,Z 384.52,A -85,B 0,C 180,E1 -11094.852,E2 -11094.852} C_VEL
LIN {X 0,Y 397.166,Z 384.512,A -85,B 0,C 180,E1 -11097.776,E2 -11097.776} C_VEL
LIN {X 0,Y 397.083,Z 384.525,A -85,B 0,C 180,E1 -11100.883,E2 -11100.883} C_VEL
LIN {X 0,Y 397.129,Z 384.517,A -85,B 0,C 180,E1 -11104.493,E2 -11104.493} C_VEL
LIN {X 0,Y 397.105,Z 384.519,A -85,B 0,C 180,E1 -11108.275,E2 -11108.275} C_VEL
LIN {X 0,Y 397.092,Z 384.521,A -85,B 0,C 180,E1 -11110.909,E2 -11110.909} C_VEL
LIN {X 0,Y 397.105,Z 384.516,A -85,B 0,C 180,E1 -11113.649,E2 -11113.649} C_VEL
LIN {X 0,Y 397.109,Z 384.523,A -85,B 0,C 180,E1 -11116.521,E2 -11116.521} C_VEL
LIN {X 0,Y 397.118,Z 384.514,A -85,B 0,C 180,E1 -11119.552,E2 -11119.552} C_VEL
LIN {X 0,Y 397.101,Z 384.519,A -85,B 0,C 180,E1 -11122.79,E2 -11122.79} C_VEL
LIN {X 0,Y 397.123,Z 384.52,A -85,B 0,C 180,E1 -11126.282,E2 -11126.282} C_VEL
LIN {X 0,Y 397.117,Z 384.519,A -85,B 0,C 180,E1 -11130.134,E2 -11130.134} C_VEL
LIN {X 0,Y 397.199,Z 384.507,A -85,B 0,C 180,E1 -11132.61,E2 -11132.61} C_VEL
LIN {X 0,Y 397.137,Z 384.516,A -85,B 0,C 180,E1 -11135.982,E2 -11135.982} C_VEL
LIN {X 0,Y 397.159,Z 384.511,A -85,B 0,C 180,E1 -11139.698,E2 -11139.698} C_VEL
LIN {X 0,Y 397.187,Z 384.506,A -85,B 0,C 180,E1 -11142.845,E2 -11142.845} C_VEL
LIN {X 0,Y 397.233,Z 384.501,A -85,B 0,C 180,E1 -11146.703,E2 -11146.703} C_VEL
LIN {X 0,Y 397.222,Z 384.506,A -85,B 0,C 180,E1 -11149.809,E2 -11149.809} C_VEL
LIN {X 0,Y 397.369,Z 384.483,A -85,B 0,C 180,E1 -11152.888,E2 -11152.888} C_VEL
LIN {X 0,Y 397.26,Z 384.497,A -85,B 0,C 180,E1 -11154.925,E2 -11154.925} C_VEL
LIN {X 0,Y 397.455,Z 384.478,A -85,B 0,C 180,E1 -11157.973,E2 -11157.973} C_VEL
LIN {X 0,Y 397.584,Z 384.461,A -85,B 0,C 180,E1 -11160,E2 -11160} C_VEL
LIN {X 0,Y 397.381,Z 384.482,A -85,B 0,C 180,E1 -11163.041,E2 -11163.041} C_VEL
LIN {X 0,Y 397.374,Z 384.485,A -85,B 0,C 180,E1 -11166.091,E2 -11166.091} C_VEL
LIN {X 0,Y 397.245,Z 384.5,A -85,B 0,C 180,E1 -11169.162,E2 -11169.162} C_VEL
LIN {X 0,Y 397.234,Z 384.501,A -85,B 0,C 180,E1 -11172.258,E2 -11172.258} C_VEL
LIN {X 0,Y 397.185,Z 384.511,A -85,B 0,C 180,E1 -11175.392,E2 -11175.392} C_VEL
LIN {X 0,Y 397.167,Z 384.508,A -85,B 0,C 180,E1 -11178.573,E2 -11178.573} C_VEL
LIN {X 0,Y 397.113,Z 384.518,A -85,B 0,C 180,E1 -11181.818,E2 -11181.818} C_VEL
LIN {X 0,Y 397.157,Z 384.515,A -85,B 0,C 180,E1 -11185.512,E2 -11185.512} C_VEL
LIN {X 0,Y 397.126,Z 384.514,A -85,B 0,C 180,E1 -11188.543,E2 -11188.543} C_VEL
LIN {X 0,Y 397.082,Z 384.519,A -85,B 0,C 180,E1 -11192.071,E2 -11192.071} C_VEL
LIN {X 0,Y 397.122,Z 384.518,A -85,B 0,C 180,E1 -11195.503,E2 -11195.503} C_VEL
LIN {X 0,Y 397.132,Z 384.516,A -85,B 0,C 180,E1 -11198.861,E2 -11198.861} C_VEL
LIN {X 0,Y 397.074,Z 384.52,A -85,B 0,C 180,E1 -11202.267,E2 -11202.267} C_VEL
LIN {X 0,Y 397.093,Z 384.524,A -85,B 0,C 180,E1 -11205.068,E2 -11205.068} C_VEL
LIN {X 0,Y 397.069,Z 384.52,A -85,B 0,C 180,E1 -11208.021,E2 -11208.021} C_VEL
LIN {X 0,Y 397.134,Z 384.518,A -85,B 0,C 180,E1 -11211.138,E2 -11211.138} C_VEL
LIN {X 0,Y 397.122,Z 384.516,A -85,B 0,C 180,E1 -11214.496,E2 -11214.496} C_VEL
LIN {X 0,Y 397.081,Z 384.519,A -85,B 0,C 180,E1 -11217.928,E2 -11217.928} C_VEL
LIN {X 0,Y 397.13,Z 384.518,A -85,B 0,C 180,E1 -11221.457,E2 -11221.457} C_VEL
LIN {X 0,Y 397.199,Z 384.719,A -85,B 0,C 180,E1 -11221.998,E2 -11221.998} C_VEL
LIN {X 0,Y 400.014,Z 398.528,A -85,B 0,C 180,E1 -11225.323,E2 -11225.323} C_VEL
LIN {X 0,Y 400.388,Z 402.32,A -85,B 0,C 180,E1 -11226.189,E2 -11226.189} C_VEL
LIN {X 0,Y 399.13,Z 418.335,A -85,B 0,C 180,E1 -11229.649,E2 -11229.649} C_VEL
LIN {X 0,Y 399.05,Z 419.741,A -85,B 0,C 180,E1 -11229.914,E2 -11229.914} C_VEL
LIN {X 0,Y 403.665,Z 447.587,A -85,B 0,C 180,E1 -11230.666,E2 -11230.666} C_VEL
LIN {X 0,Y 402.584,Z 527.617,A -85,B 0,C 180,E1 -11232.113,E2 -11232.113} C_VEL
LIN {X 0,Y 402.116,Z 540.093,A -85,B 0,C 180,E1 -11232.518,E2 -11232.518} C_VEL
LIN {X 0,Y 401.324,Z 552.997,A -85,B 0,C 180,E1 -11233.139,E2 -11233.139} C_VEL
LIN {X 0,Y 400.499,Z 565.25,A -85,B 0,C 180,E1 -11233.955,E2 -11233.955} C_VEL
LIN {X 0,Y 399.546,Z 577.095,A -85,B 0,C 180,E1 -11234.988,E2 -11234.988} C_VEL
LIN {X 0,Y 398.738,Z 587.361,A -85,B 0,C 180,E1 -11236.115,E2 -11236.115} C_VEL
LIN {X 0,Y 398.08,Z 595.803,A -85,B 0,C 180,E1 -11237.251,E2 -11237.251} C_VEL
LIN {X 0,Y 397.364,Z 603.673,A -85,B 0,C 180,E1 -11238.523,E2 -11238.523} C_VEL
LIN {X 0,Y 396.696,Z 611.361,A -85,B 0,C 180,E1 -11240.053,E2 -11240.053} C_VEL
LIN {X 0,Y 396.229,Z 618.451,A -85,B 0,C 180,E1 -11241.842,E2 -11241.842} C_VEL
LIN {X 0,Y 395.938,Z 623.169,A -85,B 0,C 180,E1 -11243.375,E2 -11243.375} C_VEL
LIN {X 0,Y 395.854,Z 626.774,A -85,B 0,C 180,E1 -11244.907,E2 -11244.907} C_VEL
LIN {X 0,Y 395.766,Z 628.633,A -85,B 0,C 180,E1 -11245.927,E2 -11245.927} C_VEL
LIN {X 0,Y 395.759,Z 631.023,A -85,B 0,C 180,E1 -11247.964,E2 -11247.964} C_VEL
LIN {X 0,Y 395.777,Z 631.63,A -85,B 0,C 180,E1 -11248.982,E2 -11248.982} C_VEL
LIN {X 0,Y 395.76,Z 631.845,A -85,B 0,C 180,E1 -11250,E2 -11250} C_VEL
LIN {X 0,Y 395.777,Z 631.628,A -85,B 0,C 180,E1 -11251.017,E2 -11251.017} C_VEL
LIN {X 0,Y 395.759,Z 631.02,A -85,B 0,C 180,E1 -11252.035,E2 -11252.035} C_VEL
LIN {X 0,Y 395.766,Z 628.626,A -85,B 0,C 180,E1 -11254.073,E2 -11254.073} C_VEL
LIN {X 0,Y 395.838,Z 625.182,A -85,B 0,C 180,E1 -11255.821,E2 -11255.821} C_VEL
LIN {X 0,Y 396.093,Z 620.123,A -85,B 0,C 180,E1 -11257.647,E2 -11257.647} C_VEL
LIN {X 0,Y 396.449,Z 614.596,A -85,B 0,C 180,E1 -11259.18,E2 -11259.18} C_VEL
LIN {X 0,Y 396.995,Z 607.697,A -85,B 0,C 180,E1 -11260.712,E2 -11260.712} C_VEL
LIN {X 0,Y 397.788,Z 599.068,A -85,B 0,C 180,E1 -11262.24,E2 -11262.24} C_VEL
LIN {X 0,Y 398.504,Z 590.286,A -85,B 0,C 180,E1 -11263.504,E2 -11263.504} C_VEL
LIN {X 0,Y 399.329,Z 579.797,A -85,B 0,C 180,E1 -11264.733,E2 -11264.733} C_VEL
LIN {X 0,Y 400.131,Z 569.875,A -85,B 0,C 180,E1 -11265.667,E2 -11265.667} C_VEL
LIN {X 0,Y 400.988,Z 557.999,A -85,B 0,C 180,E1 -11266.547,E2 -11266.547} C_VEL
LIN {X 0,Y 401.779,Z 545.643,A -85,B 0,C 180,E1 -11267.234,E2 -11267.234} C_VEL
LIN {X 0,Y 402.351,Z 532.947,A -85,B 0,C 180,E1 -11267.733,E2 -11267.733} C_VEL
LIN {X 0,Y 402.793,Z 519.63,A -85,B 0,C 180,E1 -11268.041,E2 -11268.041} C_VEL
LIN {X 0,Y 403.501,Z 446.253,A -85,B 0,C 180,E1 -11269.358,E2 -11269.358} C_VEL
LIN {X 0,Y 399.035,Z 419.507,A -85,B 0,C 180,E1 -11270.086,E2 -11270.086} C_VEL
LIN {X 0,Y 400.4,Z 402.266,A -85,B 0,C 180,E1 -11273.81,E2 -11273.81} C_VEL
LIN {X 0,Y 399.571,Z 396.065,A -85,B 0,C 180,E1 -11275.245,E2 -11275.245} C_VEL
LIN {X 0,Y 397.179,Z 384.513,A -85,B 0,C 180,E1 -11278.056,E2 -11278.056} C_VEL
LIN {X 0,Y 397.081,Z 384.523,A -85,B 0,C 180,E1 -11280.882,E2 -11280.882} C_VEL
LIN {X 0,Y 397.127,Z 384.514,A -85,B 0,C 180,E1 -11284.493,E2 -11284.493} C_VEL
LIN {X 0,Y 397.105,Z 384.516,A -85,B 0,C 180,E1 -11288.275,E2 -11288.275} C_VEL
LIN {X 0,Y 397.09,Z 384.524,A -85,B 0,C 180,E1 -11290.909,E2 -11290.909} C_VEL
LIN {X 0,Y 397.103,Z 384.517,A -85,B 0,C 180,E1 -11293.648,E2 -11293.648} C_VEL
LIN {X 0,Y 397.106,Z 384.519,A -85,B 0,C 180,E1 -11296.52,E2 -11296.52} C_VEL
LIN {X 0,Y 397.115,Z 384.517,A -85,B 0,C 180,E1 -11300.423,E2 -11300.423} C_VEL
LIN {X 0,Y 397.11,Z 384.517,A -85,B 0,C 180,E1 -11304.265,E2 -11304.265} C_VEL
LIN {X 0,Y 397.116,Z 384.522,A -85,B 0,C 180,E1 -11306.727,E2 -11306.727} C_VEL
LIN {X 0,Y 397.126,Z 384.516,A -85,B 0,C 180,E1 -11310.296,E2 -11310.296} C_VEL
LIN {X 0,Y 397.196,Z 384.511,A -85,B 0,C 180,E1 -11312.61,E2 -11312.61} C_VEL
LIN {X 0,Y 397.134,Z 384.513,A -85,B 0,C 180,E1 -11315.982,E2 -11315.982} C_VEL
LIN {X 0,Y 397.141,Z 384.512,A -85,B 0,C 180,E1 -11319.705,E2 -11319.705} C_VEL
LIN {X 0,Y 397.184,Z 384.509,A -85,B 0,C 180,E1 -11322.845,E2 -11322.845} C_VEL
LIN {X 0,Y 397.229,Z 384.505,A -85,B 0,C 180,E1 -11326.679,E2 -11326.679} C_VEL
LIN {X 0,Y 397.23,Z 384.502,A -85,B 0,C 180,E1 -11329.809,E2 -11329.809} C_VEL
LIN {X 0,Y 397.339,Z 384.488,A -85,B 0,C 180,E1 -11332.888,E2 -11332.888} C_VEL
LIN {X 0,Y 397.255,Z 384.498,A -85,B 0,C 180,E1 -11334.925,E2 -11334.925} C_VEL
LIN {X 0,Y 397.452,Z 384.477,A -85,B 0,C 180,E1 -11337.973,E2 -11337.973} C_VEL
LIN {X 0,Y 397.582,Z 384.461,A -85,B 0,C 180,E1 -11340,E2 -11340} C_VEL
LIN {X 0,Y 397.384,Z 384.481,A -85,B 0,C 180,E1 -11343.041,E2 -11343.041} C_VEL
LIN {X 0,Y 397.367,Z 384.483,A -85,B 0,C 180,E1 -11347.112,E2 -11347.112} C_VEL
LIN {X 0,Y 397.22,Z 384.507,A -85,B 0,C 180,E1 -11350.191,E2 -11350.191} C_VEL
LIN {X 0,Y 397.229,Z 384.501,A -85,B 0,C 180,E1 -11353.321,E2 -11353.321} C_VEL
LIN {X 0,Y 397.184,Z 384.506,A -85,B 0,C 180,E1 -11357.155,E2 -11357.155} C_VEL
LIN {X 0,Y 397.129,Z 384.513,A -85,B 0,C 180,E1 -11360.729,E2 -11360.729} C_VEL
LIN {X 0,Y 397.135,Z 384.517,A -85,B 0,C 180,E1 -11364.018,E2 -11364.018} C_VEL
LIN {X 0,Y 397.197,Z 384.507,A -85,B 0,C 180,E1 -11367.39,E2 -11367.39} C_VEL
LIN {X 0,Y 397.085,Z 384.518,A -85,B 0,C 180,E1 -11370.882,E2 -11370.882} C_VEL
LIN {X 0,Y 397.128,Z 384.513,A -85,B 0,C 180,E1 -11374.493,E2 -11374.493} C_VEL
LIN {X 0,Y 397.109,Z 384.516,A -85,B 0,C 180,E1 -11378.275,E2 -11378.275} C_VEL
LIN {X 0,Y 397.109,Z 384.516,A -85,B 0,C 180,E1 -11380.906,E2 -11380.906} C_VEL
LIN {X 0,Y 397.106,Z 384.522,A -85,B 0,C 180,E1 -11383.648,E2 -11383.648} C_VEL
LIN {X 0,Y 397.104,Z 384.516,A -85,B 0,C 180,E1 -11386.521,E2 -11386.521} C_VEL
LIN {X 0,Y 397.116,Z 384.515,A -85,B 0,C 180,E1 -11390.423,E2 -11390.423} C_VEL
LIN {X 0,Y 397.112,Z 384.515,A -85,B 0,C 180,E1 -11394.266,E2 -11394.266} C_VEL
LIN {X 0,Y 397.117,Z 384.516,A -85,B 0,C 180,E1 -11396.727,E2 -11396.727} C_VEL
LIN {X 0,Y 397.127,Z 384.513,A -85,B 0,C 180,E1 -11400.296,E2 -11400.296} C_VEL
LIN {X 0,Y 397.197,Z 384.505,A -85,B 0,C 180,E1 -11402.61,E2 -11402.61} C_VEL
LIN {X 0,Y 397.17,Z 384.602,A -85,B 0,C 180,E1 -11405.323,E2 -11405.323} C_VEL
LIN {X 0,Y 399.344,Z 395.741,A -85,B 0,C 180,E1 -11408.311,E2 -11408.311} C_VEL
LIN {X 0,Y 399.515,Z 400.096,A -85,B 0,C 180,E1 -11409.401,E2 -11409.401} C_VEL
LIN {X 0,Y 399.313,Z 402.504,A -85,B 0,C 180,E1 -11409.983,E2 -11409.983} C_VEL
LIN {X 0,Y 403.899,Z 425.689,A -85,B 0,C 180,E1 -11410.658,E2 -11410.658} C_VEL
LIN {X 0,Y 402.762,Z 510.017,A -85,B 0,C 180,E1 -11412.187,E2 -11412.187} C_VEL
LIN {X 0,Y 402.208,Z 523.839,A -85,B 0,C 180,E1 -11412.654,E2 -11412.654} C_VEL
LIN {X 0,Y 401.565,Z 536.22,A -85,B 0,C 180,E1 -11413.281,E2 -11413.281} C_VEL
LIN {X 0,Y 400.834,Z 548.063,A -85,B 0,C 180,E1 -11414.1,E2 -11414.1} C_VEL
LIN {X 0,Y 400.044,Z 559.814,A -85,B 0,C 180,E1 -11415.151,E2 -11415.151} C_VEL
LIN {X 0,Y 399.244,Z 569.662,A -85,B 0,C 180,E1 -11416.253,E2 -11416.253} C_VEL
LIN {X 0,Y 398.442,Z 578.849,A -85,B 0,C 180,E1 -11417.522,E2 -11417.522} C_VEL
LIN {X 0,Y 397.588,Z 587.77,A -85,B 0,C 180,E1 -11419.046,E2 -11419.046} C_VEL
LIN {X 0,Y 396.976,Z 594.951,A -85,B 0,C 180,E1 -11420.575,E2 -11420.575} C_VEL
LIN {X 0,Y 396.533,Z 599.795,A -85,B 0,C 180,E1 -11421.849,E2 -11421.849} C_VEL
LIN {X 0,Y 396.239,Z 604.405,A -85,B 0,C 180,E1 -11423.346,E2 -11423.346} C_VEL
LIN {X 0,Y 396.045,Z 608.101,A -85,B 0,C 180,E1 -11424.91,E2 -11424.91} C_VEL
LIN {X 0,Y 395.867,Z 609.964,A -85,B 0,C 180,E1 -11425.928,E2 -11425.928} C_VEL
LIN {X 0,Y 395.837,Z 611.365,A -85,B 0,C 180,E1 -11426.947,E2 -11426.947} C_VEL
LIN {X 0,Y 395.841,Z 612.36,A -85,B 0,C 180,E1 -11427.965,E2 -11427.965} C_VEL
LIN {X 0,Y 395.761,Z 613.209,A -85,B 0,C 180,E1 -11430,E2 -11430} C_VEL
LIN {X 0,Y 395.796,Z 613.019,A -85,B 0,C 180,E1 -11431.018,E2 -11431.018} C_VEL
LIN {X 0,Y 395.841,Z 612.434,A -85,B 0,C 180,E1 -11432.035,E2 -11432.035} C_VEL
LIN {X 0,Y 395.863,Z 610.128,A -85,B 0,C 180,E1 -11434.06,E2 -11434.06} C_VEL
LIN {X 0,Y 395.277,Z 608.87,A -85,B 0,C 180,E1 -11434.893,E2 -11434.893} C_VEL
LIN {X 0,Y 392.579,Z 606.211,A -85,B 0,C 180,E1 -11436.228,E2 -11436.228} C_VEL
LIN {X 0,Y 390.35,Z 603.506,A -85,B 0,C 180,E1 -11437.279,E2 -11437.279} C_VEL
LIN {X 0,Y 389.502,Z 601.088,A -85,B 0,C 180,E1 -11438.067,E2 -11438.067} C_VEL
LIN {X 0,Y 389.493,Z 600.206,A -85,B 0,C 180,E1 -11438.328,E2 -11438.328} C_VEL
LIN {X 0,Y 390.118,Z 593.313,A -85,B 0,C 180,E1 -11440.117,E2 -11440.117} C_VEL
LIN {X 0,Y 390.873,Z 585.74,A -85,B 0,C 180,E1 -11441.67,E2 -11441.67} C_VEL
LIN {X 0,Y 391.589,Z 577.982,A -85,B 0,C 180,E1 -11442.964,E2 -11442.964} C_VEL
LIN {X 0,Y 392.569,Z 567.434,A -85,B 0,C 180,E1 -11444.383,E2 -11444.383} C_VEL
LIN {X 0,Y 393.366,Z 556.687,A -85,B 0,C 180,E1 -11445.545,E2 -11445.545} C_VEL
LIN {X 0,Y 394.167,Z 546.208,A -85,B 0,C 180,E1 -11446.443,E2 -11446.443} C_VEL
LIN {X 0,Y 395.028,Z 533.583,A -85,B 0,C 180,E1 -11447.271,E2 -11447.271} C_VEL
LIN {X 0,Y 395.625,Z 520.948,A -85,B 0,C 180,E1 -11447.878,E2 -11447.878} C_VEL
LIN {X 0,Y 396.045,Z 508.959,A -85,B 0,C 180,E1 -11448.26,E2 -11448.26} C_VEL
LIN {X 0,Y 397.05,Z 434.994,A -85,B 0,C 180,E1 -11449.617,E2 -11449.617} C_VEL
LIN {X 0,Y 397.034,Z 425.309,A -85,B 0,C 180,E1 -11449.8,E2 -11449.8} C_VEL
LIN {X 0,Y 392.489,Z 402.552,A -85,B 0,C 180,E1 -11450.506,E2 -11450.506} C_VEL
LIN {X 0,Y 392.534,Z 397.877,A -85,B 0,C 180,E1 -11451.684,E2 -11451.684} C_VEL
LIN {X 0,Y 390.137,Z 385.409,A -85,B 0,C 180,E1 -11455.081,E2 -11455.081} C_VEL
LIN {X 0,Y 390.1,Z 385.391,A -85,B 0,C 180,E1 -11458.02,E2 -11458.02} C_VEL
LIN {X 0,Y 390.027,Z 385.398,A -85,B 0,C 180,E1 -11461.504,E2 -11461.504} C_VEL
LIN {X 0,Y 390.089,Z 385.392,A -85,B 0,C 180,E1 -11465.207,E2 -11465.207} C_VEL
LIN {X 0,Y 390.072,Z 385.393,A -85,B 0,C 180,E1 -11469.218,E2 -11469.218} C_VEL
LIN {X 0,Y 390.046,Z 385.4,A -85,B 0,C 180,E1 -11472.374,E2 -11472.374} C_VEL
LIN {X 0,Y 390.05,Z 385.395,A -85,B 0,C 180,E1 -11475.355,E2 -11475.355} C_VEL
LIN {X 0,Y 390.048,Z 385.398,A -85,B 0,C 180,E1 -11478.189,E2 -11478.189} C_VEL
LIN {X 0,Y 390.096,Z 385.391,A -85,B 0,C 180,E1 -11480.908,E2 -11480.908} C_VEL
LIN {X 0,Y 390.089,Z 385.393,A -85,B 0,C 180,E1 -11484.793,E2 -11484.793} C_VEL
LIN {X 0,Y 390.031,Z 385.402,A -85,B 0,C 180,E1 -11488.496,E2 -11488.496} C_VEL
LIN {X 0,Y 390.121,Z 385.39,A -85,B 0,C 180,E1 -11492.07,E2 -11492.07} C_VEL
LIN {X 0,Y 390.084,Z 385.391,A -85,B 0,C 180,E1 -11495.519,E2 -11495.519} C_VEL
LIN {X 0,Y 390.077,Z 385.392,A -85,B 0,C 180,E1 -11498.879,E2 -11498.879} C_VEL
LIN {X 0,Y 390.136,Z 385.391,A -85,B 0,C 180,E1 -11502.167,E2 -11502.167} C_VEL
LIN {X 0,Y 390.149,Z 385.383,A -85,B 0,C 180,E1 -11505.393,E2 -11505.393} C_VEL
LIN {X 0,Y 390.153,Z 385.383,A -85,B 0,C 180,E1 -11508.571,E2 -11508.571} C_VEL
LIN {X 0,Y 390.349,Z 385.364,A -85,B 0,C 180,E1 -11511.993,E2 -11511.993} C_VEL
LIN {X 0,Y 390.232,Z 385.372,A -85,B 0,C 180,E1 -11514.834,E2 -11514.834} C_VEL
LIN {X 0,Y 390.423,Z 385.354,A -85,B 0,C 180,E1 -11517.937,E2 -11517.937} C_VEL
LIN {X 0,Y 390.554,Z 385.337,A -85,B 0,C 180,E1 -11520,E2 -11520} C_VEL
LIN {X 0,Y 390.316,Z 385.362,A -85,B 0,C 180,E1 -11523.096,E2 -11523.096} C_VEL
LIN {X 0,Y 390.326,Z 385.362,A -85,B 0,C 180,E1 -11526.202,E2 -11526.202} C_VEL
LIN {X 0,Y 390.202,Z 385.379,A -85,B 0,C 180,E1 -11529.329,E2 -11529.329} C_VEL
LIN {X 0,Y 390.183,Z 385.378,A -85,B 0,C 180,E1 -11532.483,E2 -11532.483} C_VEL
LIN {X 0,Y 390.145,Z 385.389,A -85,B 0,C 180,E1 -11535.677,E2 -11535.677} C_VEL
LIN {X 0,Y 390.11,Z 385.388,A -85,B 0,C 180,E1 -11538.922,E2 -11538.922} C_VEL
LIN {X 0,Y 390.051,Z 385.395,A -85,B 0,C 180,E1 -11542.233,E2 -11542.233} C_VEL
LIN {X 0,Y 390.123,Z 385.389,A -85,B 0,C 180,E1 -11545.743,E2 -11545.743} C_VEL
LIN {X 0,Y 390.063,Z 385.397,A -85,B 0,C 180,E1 -11549.109,E2 -11549.109} C_VEL
LIN {X 0,Y 390.047,Z 385.396,A -85,B 0,C 180,E1 -11552.721,E2 -11552.721} C_VEL
LIN {X 0,Y 390.059,Z 385.395,A -85,B 0,C 180,E1 -11555.825,E2 -11555.825} C_VEL
LIN {X 0,Y 390.072,Z 385.399,A -85,B 0,C 180,E1 -11559.218,E2 -11559.218} C_VEL
LIN {X 0,Y 390.047,Z 385.396,A -85,B 0,C 180,E1 -11562.374,E2 -11562.374} C_VEL
LIN {X 0,Y 390.05,Z 385.399,A -85,B 0,C 180,E1 -11565.354,E2 -11565.354} C_VEL
LIN {X 0,Y 390.034,Z 385.397,A -85,B 0,C 180,E1 -11568.187,E2 -11568.187} C_VEL
LIN {X 0,Y 390.094,Z 385.395,A -85,B 0,C 180,E1 -11570.908,E2 -11570.908} C_VEL
LIN {X 0,Y 390.088,Z 385.395,A -85,B 0,C 180,E1 -11574.793,E2 -11574.793} C_VEL
LIN {X 0,Y 390.027,Z 385.4,A -85,B 0,C 180,E1 -11578.496,E2 -11578.496} C_VEL
LIN {X 0,Y 390.114,Z 385.485,A -85,B 0,C 180,E1 -11581.661,E2 -11581.661} C_VEL
LIN {X 0,Y 392.549,Z 397.184,A -85,B 0,C 180,E1 -11584.552,E2 -11584.552} C_VEL
LIN {X 0,Y 393.469,Z 403.403,A -85,B 0,C 180,E1 -11586.024,E2 -11586.024} C_VEL
LIN {X 0,Y 392.195,Z 419.093,A -85,B 0,C 180,E1 -11589.479,E2 -11589.479} C_VEL
LIN {X 0,Y 392.273,Z 420.223,A -85,B 0,C 180,E1 -11589.564,E2 -11589.564} C_VEL
LIN {X 0,Y 396.959,Z 448.312,A -85,B 0,C 180,E1 -11590.343,E2 -11590.343} C_VEL
LIN {X 0,Y 395.851,Z 527.463,A -85,B 0,C 180,E1 -11591.798,E2 -11591.798} C_VEL
LIN {X 0,Y 395.368,Z 539.934,A -85,B 0,C 180,E1 -11592.21,E2 -11592.21} C_VEL
LIN {X 0,Y 394.533,Z 552.836,A -85,B 0,C 180,E1 -11592.84,E2 -11592.84} C_VEL
LIN {X 0,Y 393.659,Z 565.087,A -85,B 0,C 180,E1 -11593.669,E2 -11593.669} C_VEL
LIN {X 0,Y 392.666,Z 576.931,A -85,B 0,C 180,E1 -11594.719,E2 -11594.719} C_VEL
LIN {X 0,Y 391.829,Z 587.273,A -85,B 0,C 180,E1 -11595.875,E2 -11595.875} C_VEL
LIN {X 0,Y 391.138,Z 595.638,A -85,B 0,C 180,E1 -11597.02,E2 -11597.02} C_VEL
LIN {X 0,Y 390.359,Z 603.507,A -85,B 0,C 180,E1 -11598.314,E2 -11598.314} C_VEL
LIN {X 0,Y 389.678,Z 611.194,A -85,B 0,C 180,E1 -11599.872,E2 -11599.872} C_VEL
LIN {X 0,Y 389.186,Z 618.285,A -85,B 0,C 180,E1 -11601.693,E2 -11601.693} C_VEL
LIN {X 0,Y 388.853,Z 623.001,A -85,B 0,C 180,E1 -11603.253,E2 -11603.253} C_VEL
LIN {X 0,Y 388.75,Z 626.607,A -85,B 0,C 180,E1 -11604.814,E2 -11604.814} C_VEL
LIN {X 0,Y 388.693,Z 628.466,A -85,B 0,C 180,E1 -11605.852,E2 -11605.852} C_VEL
LIN {X 0,Y 388.657,Z 630.855,A -85,B 0,C 180,E1 -11607.927,E2 -11607.927} C_VEL
LIN {X 0,Y 388.69,Z 631.464,A -85,B 0,C 180,E1 -11608.964,E2 -11608.964} C_VEL
LIN {X 0,Y 388.69,Z 631.679,A -85,B 0,C 180,E1 -11610,E2 -11610} C_VEL
LIN {X 0,Y 388.69,Z 631.461,A -85,B 0,C 180,E1 -11611.036,E2 -11611.036} C_VEL
LIN {X 0,Y 388.657,Z 630.852,A -85,B 0,C 180,E1 -11612.072,E2 -11612.072} C_VEL
LIN {X 0,Y 388.693,Z 628.459,A -85,B 0,C 180,E1 -11614.147,E2 -11614.147} C_VEL
LIN {X 0,Y 388.738,Z 625.385,A -85,B 0,C 180,E1 -11615.77,E2 -11615.77} C_VEL
LIN {X 0,Y 388.942,Z 621.548,A -85,B 0,C 180,E1 -11617.266,E2 -11617.266} C_VEL
LIN {X 0,Y 389.354,Z 615.439,A -85,B 0,C 180,E1 -11619.087,E2 -11619.087} C_VEL
LIN {X 0,Y 389.889,Z 608.764,A -85,B 0,C 180,E1 -11620.647,E2 -11620.647} C_VEL
LIN {X 0,Y 390.682,Z 600.486,A -85,B 0,C 180,E1 -11622.203,E2 -11622.203} C_VEL
LIN {X 0,Y 391.411,Z 591.997,A -85,B 0,C 180,E1 -11623.498,E2 -11623.498} C_VEL
LIN {X 0,Y 392.289,Z 581.508,A -85,B 0,C 180,E1 -11624.791,E2 -11624.791} C_VEL
LIN {X 0,Y 393.163,Z 571.132,A -85,B 0,C 180,E1 -11625.819,E2 -11625.819} C_VEL
LIN {X 0,Y 394.053,Z 559.755,A -85,B 0,C 180,E1 -11626.714,E2 -11626.714} C_VEL
LIN {X 0,Y 394.835,Z 548.071,A -85,B 0,C 180,E1 -11627.413,E2 -11627.413} C_VEL
LIN {X 0,Y 395.541,Z 534.603,A -85,B 0,C 180,E1 -11627.982,E2 -11627.982} C_VEL
LIN {X 0,Y 396.019,Z 521.233,A -85,B 0,C 180,E1 -11628.327,E2 -11628.327} C_VEL
LIN {X 0,Y 396.821,Z 447.216,A -85,B 0,C 180,E1 -11629.676,E2 -11629.676} C_VEL
LIN {X 0,Y 392.144,Z 419.344,A -85,B 0,C 180,E1 -11630.455,E2 -11630.455} C_VEL
LIN {X 0,Y 393.409,Z 404.585,A -85,B 0,C 180,E1 -11633.7,E2 -11633.7} C_VEL
LIN {X 0,Y 393.212,Z 400.863,A -85,B 0,C 180,E1 -11634.554,E2 -11634.554} C_VEL
LIN {X 0,Y 391.034,Z 389.668,A -85,B 0,C 180,E1 -11637.278,E2 -11637.278} C_VEL
LIN {X 0,Y 390.095,Z 385.395,A -85,B 0,C 180,E1 -11638.377,E2 -11638.377} C_VEL
LIN {X 0,Y 390.033,Z 385.397,A -85,B 0,C 180,E1 -11642.125,E2 -11642.125} C_VEL
LIN {X 0,Y 390.087,Z 385.396,A -85,B 0,C 180,E1 -11645.207,E2 -11645.207} C_VEL
LIN {X 0,Y 390.072,Z 385.396,A -85,B 0,C 180,E1 -11649.218,E2 -11649.218} C_VEL
LIN {X 0,Y 390.044,Z 385.397,A -85,B 0,C 180,E1 -11652.374,E2 -11652.374} C_VEL
LIN {X 0,Y 390.048,Z 385.397,A -85,B 0,C 180,E1 -11655.355,E2 -11655.355} C_VEL
LIN {X 0,Y 390.034,Z 385.397,A -85,B 0,C 180,E1 -11658.187,E2 -11658.187} C_VEL
LIN {X 0,Y 390.092,Z 385.396,A -85,B 0,C 180,E1 -11660.908,E2 -11660.908} C_VEL
LIN {X 0,Y 390.087,Z 385.397,A -85,B 0,C 180,E1 -11664.793,E2 -11664.793} C_VEL
LIN {X 0,Y 390.026,Z 385.402,A -85,B 0,C 180,E1 -11668.496,E2 -11668.496} C_VEL
LIN {X 0,Y 390.119,Z 385.387,A -85,B 0,C 180,E1 -11672.07,E2 -11672.07} C_VEL
LIN {X 0,Y 390.081,Z 385.391,A -85,B 0,C 180,E1 -11675.519,E2 -11675.519} C_VEL
LIN {X 0,Y 390.065,Z 385.396,A -85,B 0,C 180,E1 -11678.878,E2 -11678.878} C_VEL
LIN {X 0,Y 390.13,Z 385.388,A -85,B 0,C 180,E1 -11682.167,E2 -11682.167} C_VEL
LIN {X 0,Y 390.149,Z 385.382,A -85,B 0,C 180,E1 -11685.393,E2 -11685.393} C_VEL
LIN {X 0,Y 390.161,Z 385.386,A -85,B 0,C 180,E1 -11688.572,E2 -11688.572} C_VEL
LIN {X 0,Y 390.272,Z 385.371,A -85,B 0,C 180,E1 -11692.071,E2 -11692.071} C_VEL
LIN {X 0,Y 390.227,Z 385.374,A -85,B 0,C 180,E1 -11694.834,E2 -11694.834} C_VEL
LIN {X 0,Y 390.421,Z 385.352,A -85,B 0,C 180,E1 -11697.937,E2 -11697.937} C_VEL
LIN {X 0,Y 390.551,Z 385.337,A -85,B 0,C 180,E1 -11700,E2 -11700} C_VEL
LIN {X 0,Y 390.318,Z 385.361,A -85,B 0,C 180,E1 -11703.097,E2 -11703.097} C_VEL
LIN {X 0,Y 390.312,Z 385.364,A -85,B 0,C 180,E1 -11706.642,E2 -11706.642} C_VEL
LIN {X 0,Y 390.207,Z 385.376,A -85,B 0,C 180,E1 -11709.329,E2 -11709.329} C_VEL
LIN {X 0,Y 390.197,Z 385.378,A -85,B 0,C 180,E1 -11713.438,E2 -11713.438} C_VEL
LIN {X 0,Y 390.151,Z 385.383,A -85,B 0,C 180,E1 -11717.308,E2 -11717.308} C_VEL
LIN {X 0,Y 390.104,Z 385.389,A -85,B 0,C 180,E1 -11720.476,E2 -11720.476} C_VEL
LIN {X 0,Y 390.092,Z 385.391,A -85,B 0,C 180,E1 -11723.351,E2 -11723.351} C_VEL
LIN {X 0,Y 390.116,Z 385.387,A -85,B 0,C 180,E1 -11726.768,E2 -11726.768} C_VEL
LIN {X 0,Y 390.045,Z 385.397,A -85,B 0,C 180,E1 -11730.299,E2 -11730.299} C_VEL
LIN {X 0,Y 390.07,Z 385.395,A -85,B 0,C 180,E1 -11734.025,E2 -11734.025} C_VEL
LIN {X 0,Y 390.048,Z 385.401,A -85,B 0,C 180,E1 -11737.551,E2 -11737.551} C_VEL
LIN {X 0,Y 390.074,Z 385.392,A -85,B 0,C 180,E1 -11740.824,E2 -11740.824} C_VEL
LIN {X 0,Y 390.059,Z 385.397,A -85,B 0,C 180,E1 -11743.887,E2 -11743.887} C_VEL
LIN {X 0,Y 390.059,Z 385.394,A -85,B 0,C 180,E1 -11746.79,E2 -11746.79} C_VEL
LIN {X 0,Y 390.058,Z 385.399,A -85,B 0,C 180,E1 -11749.561,E2 -11749.561} C_VEL
LIN {X 0,Y 390.047,Z 385.395,A -85,B 0,C 180,E1 -11752.449,E2 -11752.449} C_VEL
LIN {X 0,Y 390.086,Z 385.391,A -85,B 0,C 180,E1 -11756.047,E2 -11756.047} C_VEL
LIN {X 0,Y 390.049,Z 385.396,A -85,B 0,C 180,E1 -11759.869,E2 -11759.869} C_VEL
LIN {X 0,Y 390.116,Z 385.394,A -85,B 0,C 180,E1 -11763.232,E2 -11763.232} C_VEL
LIN {X 0,Y 390.134,Z 385.431,A -85,B 0,C 180,E1 -11765.026,E2 -11765.026} C_VEL
LIN {X 0,Y 392.468,Z 397.525,A -85,B 0,C 180,E1 -11768.322,E2 -11768.322} C_VEL
LIN {X 0,Y 392.477,Z 402.693,A -85,B 0,C 180,E1 -11769.625,E2 -11769.625} C_VEL
LIN {X 0,Y 397.073,Z 425.525,A -85,B 0,C 180,E1 -11770.305,E2 -11770.305} C_VEL
LIN {X 0,Y 396.176,Z 501.121,A -85,B 0,C 180,E1 -11771.68,E2 -11771.68} C_VEL
LIN {X 0,Y 395.906,Z 514.712,A -85,B 0,C 180,E1 -11772.002,E2 -11772.002} C_VEL
LIN {X 0,Y 395.34,Z 526.85,A -85,B 0,C 180,E1 -11772.476,E2 -11772.476} C_VEL
LIN {X 0,Y 394.597,Z 539.382,A -85,B 0,C 180,E1 -11773.177,E2 -11773.177} C_VEL
LIN {X 0,Y 393.788,Z 551.385,A -85,B 0,C 180,E1 -11774.074,E2 -11774.074} C_VEL
LIN {X 0,Y 393.052,Z 562.095,A -85,B 0,C 180,E1 -11775.109,E2 -11775.109} C_VEL
LIN {X 0,Y 392.209,Z 571.791,A -85,B 0,C 180,E1 -11776.265,E2 -11776.265} C_VEL
LIN {X 0,Y 391.296,Z 580.641,A -85,B 0,C 180,E1 -11777.554,E2 -11777.554} C_VEL
LIN {X 0,Y 390.471,Z 589.272,A -85,B 0,C 180,E1 -11779.106,E2 -11779.106} C_VEL
LIN {X 0,Y 389.859,Z 596.151,A -85,B 0,C 180,E1 -11780.663,E2 -11780.663} C_VEL
LIN {X 0,Y 389.374,Z 601.659,A -85,B 0,C 180,E1 -11782.22,E2 -11782.22} C_VEL
LIN {X 0,Y 389.088,Z 605.982,A -85,B 0,C 180,E1 -11783.778,E2 -11783.778} C_VEL
LIN {X 0,Y 388.99,Z 608.268,A -85,B 0,C 180,E1 -11784.817,E2 -11784.817} C_VEL
LIN {X 0,Y 388.795,Z 610.131,A -85,B 0,C 180,E1 -11785.854,E2 -11785.854} C_VEL
LIN {X 0,Y 388.741,Z 611.532,A -85,B 0,C 180,E1 -11786.891,E2 -11786.891} C_VEL
LIN {X 0,Y 388.742,Z 612.528,A -85,B 0,C 180,E1 -11787.928,E2 -11787.928} C_VEL
LIN {X 0,Y 388.692,Z 613.375,A -85,B 0,C 180,E1 -11790,E2 -11790} C_VEL
LIN {X 0,Y 388.71,Z 613.186,A -85,B 0,C 180,E1 -11791.036,E2 -11791.036} C_VEL
LIN {X 0,Y 388.742,Z 612.601,A -85,B 0,C 180,E1 -11792.072,E2 -11792.072} C_VEL
LIN {X 0,Y 388.792,Z 610.278,A -85,B 0,C 180,E1 -11794.147,E2 -11794.147} C_VEL
LIN {X 0,Y 389.044,Z 607.407,A -85,B 0,C 180,E1 -11795.702,E2 -11795.702} C_VEL
LIN {X 0,Y 389.252,Z 603.519,A -85,B 0,C 180,E1 -11797.261,E2 -11797.261} C_VEL
LIN {X 0,Y 389.493,Z 600.206,A -85,B 0,C 180,E1 -11798.328,E2 -11798.328} C_VEL
LIN {X 0,Y 389.063,Z 597.533,A -85,B 0,C 180,E1 -11799.098,E2 -11799.098} C_VEL
LIN {X 0,Y 385.557,Z 590.833,A -85,B 0,C 180,E1 -11800.826,E2 -11800.826} C_VEL
LIN {X 0,Y 384.086,Z 586.411,A -85,B 0,C 180,E1 -11801.779,E2 -11801.779} C_VEL
LIN {X 0,Y 384.04,Z 583.938,A -85,B 0,C 180,E1 -11802.24,E2 -11802.24} C_VEL
LIN {X 0,Y 385.03,Z 574.596,A -85,B 0,C 180,E1 -11803.727,E2 -11803.727} C_VEL
LIN {X 0,Y 385.972,Z 564.1,A -85,B 0,C 180,E1 -11805.059,E2 -11805.059} C_VEL
LIN {X 0,Y 386.753,Z 554.041,A -85,B 0,C 180,E1 -11806.089,E2 -11806.089} C_VEL
LIN {X 0,Y 387.681,Z 542.845,A -85,B 0,C 180,E1 -11806.997,E2 -11806.997} C_VEL
LIN {X 0,Y 388.412,Z 531.484,A -85,B 0,C 180,E1 -11807.711,E2 -11807.711} C_VEL
LIN {X 0,Y 388.981,Z 518.512,A -85,B 0,C 180,E1 -11808.296,E2 -11808.296} C_VEL
LIN {X 0,Y 389.419,Z 504.619,A -85,B 0,C 180,E1 -11808.684,E2 -11808.684} C_VEL
LIN {X 0,Y 390.389,Z 426.39,A -85,B 0,C 180,E1 -11810.134,E2 -11810.134} C_VEL
LIN {X 0,Y 385.653,Z 402.716,A -85,B 0,C 180,E1 -11810.886,E2 -11810.886} C_VEL
LIN {X 0,Y 385.435,Z 398.414,A -85,B 0,C 180,E1 -11812.008,E2 -11812.008} C_VEL
LIN {X 0,Y 383.105,Z 386.272,A -85,B 0,C 180,E1 -11815.392,E2 -11815.392} C_VEL
LIN {X 0,Y 383.044,Z 386.271,A -85,B 0,C 180,E1 -11818.493,E2 -11818.493} C_VEL
LIN {X 0,Y 383.013,Z 386.272,A -85,B 0,C 180,E1 -11822.15,E2 -11822.15} C_VEL
LIN {X 0,Y 383.021,Z 386.277,A -85,B 0,C 180,E1 -11824.668,E2 -11824.668} C_VEL
LIN {X 0,Y 383.002,Z 386.273,A -85,B 0,C 180,E1 -11827.904,E2 -11827.904} C_VEL
LIN {X 0,Y 382.987,Z 386.275,A -85,B 0,C 180,E1 -11831.348,E2 -11831.348} C_VEL
LIN {X 0,Y 383.001,Z 386.277,A -85,B 0,C 180,E1 -11834.304,E2 -11834.304} C_VEL
LIN {X 0,Y 383.014,Z 386.272,A -85,B 0,C 180,E1 -11837.24,E2 -11837.24} C_VEL
LIN {X 0,Y 383.023,Z 386.276,A -85,B 0,C 180,E1 -11840.413,E2 -11840.413} C_VEL
LIN {X 0,Y 383.03,Z 386.272,A -85,B 0,C 180,E1 -11844.045,E2 -11844.045} C_VEL
LIN {X 0,Y 382.992,Z 386.274,A -85,B 0,C 180,E1 -11847.578,E2 -11847.578} C_VEL
LIN {X 0,Y 383.002,Z 386.28,A -85,B 0,C 180,E1 -11850.301,E2 -11850.301} C_VEL
LIN {X 0,Y 383.061,Z 386.268,A -85,B 0,C 180,E1 -11852.698,E2 -11852.698} C_VEL
LIN {X 0,Y 383.056,Z 386.266,A -85,B 0,C 180,E1 -11855.04,E2 -11855.04} C_VEL
LIN {X 0,Y 383.009,Z 386.275,A -85,B 0,C 180,E1 -11858.47,E2 -11858.47} C_VEL
LIN {X 0,Y 383.099,Z 386.264,A -85,B 0,C 180,E1 -11861.828,E2 -11861.828} C_VEL
LIN {X 0,Y 383.115,Z 386.259,A -85,B 0,C 180,E1 -11865.118,E2 -11865.118} C_VEL
LIN {X 0,Y 383.102,Z 386.263,A -85,B 0,C 180,E1 -11868.358,E2 -11868.358} C_VEL
LIN {X 0,Y 383.309,Z 386.241,A -85,B 0,C 180,E1 -11871.933,E2 -11871.933} C_VEL
LIN {X 0,Y 383.204,Z 386.248,A -85,B 0,C 180,E1 -11874.738,E2 -11874.738} C_VEL
LIN {X 0,Y 383.391,Z 386.231,A -85,B 0,C 180,E1 -11877.899,E2 -11877.899} C_VEL
LIN {X 0,Y 383.523,Z 386.213,A -85,B 0,C 180,E1 -11880,E2 -11880} C_VEL
LIN {X 0,Y 383.253,Z 386.243,A -85,B 0,C 180,E1 -11883.154,E2 -11883.154} C_VEL
LIN {X 0,Y 383.281,Z 386.239,A -85,B 0,C 180,E1 -11886.316,E2 -11886.316} C_VEL
LIN {X 0,Y 383.152,Z 386.259,A -85,B 0,C 180,E1 -11889.502,E2 -11889.502} C_VEL
LIN {X 0,Y 383.146,Z 386.255,A -85,B 0,C 180,E1 -11892.716,E2 -11892.716} C_VEL
LIN {X 0,Y 383.086,Z 386.265,A -85,B 0,C 180,E1 -11895.973,E2 -11895.973} C_VEL
LIN {X 0,Y 383.065,Z 386.269,A -85,B 0,C 180,E1 -11899.283,E2 -11899.283} C_VEL
LIN {X 0,Y 383.017,Z 386.271,A -85,B 0,C 180,E1 -11902.664,E2 -11902.664} C_VEL
LIN {X 0,Y 383.084,Z 386.263,A -85,B 0,C 180,E1 -11906.123,E2 -11906.123} C_VEL
LIN {X 0,Y 382.996,Z 386.276,A -85,B 0,C 180,E1 -11909.7,E2 -11909.7} C_VEL
LIN {X 0,Y 383.007,Z 386.278,A -85,B 0,C 180,E1 -11913.4,E2 -11913.4} C_VEL
LIN {X 0,Y 383.035,Z 386.269,A -85,B 0,C 180,E1 -11916.164,E2 -11916.164} C_VEL
LIN {X 0,Y 383.012,Z 386.272,A -85,B 0,C 180,E1 -11919.958,E2 -11919.958} C_VEL
LIN {X 0,Y 383.008,Z 386.275,A -85,B 0,C 180,E1 -11922.778,E2 -11922.778} C_VEL
LIN {X 0,Y 383.001,Z 386.273,A -85,B 0,C 180,E1 -11925.789,E2 -11925.789} C_VEL
LIN {X 0,Y 382.991,Z 386.278,A -85,B 0,C 180,E1 -11928.796,E2 -11928.796} C_VEL
LIN {X 0,Y 383.003,Z 386.273,A -85,B 0,C 180,E1 -11932.096,E2 -11932.096} C_VEL
LIN {X 0,Y 383.021,Z 386.273,A -85,B 0,C 180,E1 -11935.332,E2 -11935.332} C_VEL
LIN {X 0,Y 382.986,Z 386.281,A -85,B 0,C 180,E1 -11939.081,E2 -11939.081} C_VEL
LIN {X 0,Y 383.091,Z 386.444,A -85,B 0,C 180,E1 -11941.361,E2 -11941.361} C_VEL
LIN {X 0,Y 385.558,Z 398.269,A -85,B 0,C 180,E1 -11944.347,E2 -11944.347} C_VEL
LIN {X 0,Y 386.555,Z 404.658,A -85,B 0,C 180,E1 -11945.894,E2 -11945.894} C_VEL
LIN {X 0,Y 385.299,Z 419.188,A -85,B 0,C 180,E1 -11949.155,E2 -11949.155} C_VEL
LIN {X 0,Y 390.268,Z 449.067,A -85,B 0,C 180,E1 -11950.009,E2 -11950.009} C_VEL
LIN {X 0,Y 389.128,Z 527.309,A -85,B 0,C 180,E1 -11951.472,E2 -11951.472} C_VEL
LIN {X 0,Y 388.607,Z 539.775,A -85,B 0,C 180,E1 -11951.89,E2 -11951.89} C_VEL
LIN {X 0,Y 387.755,Z 552.675,A -85,B 0,C 180,E1 -11952.531,E2 -11952.531} C_VEL
LIN {X 0,Y 386.842,Z 564.924,A -85,B 0,C 180,E1 -11953.373,E2 -11953.373} C_VEL
LIN {X 0,Y 385.837,Z 576.508,A -85,B 0,C 180,E1 -11954.415,E2 -11954.415} C_VEL
LIN {X 0,Y 384.865,Z 587.704,A -85,B 0,C 180,E1 -11955.69,E2 -11955.69} C_VEL
LIN {X 0,Y 384.027,Z 597.148,A -85,B 0,C 180,E1 -11957.045,E2 -11957.045} C_VEL
LIN {X 0,Y 383.097,Z 606.077,A -85,B 0,C 180,E1 -11958.626,E2 -11958.626} C_VEL
LIN {X 0,Y 382.481,Z 613.265,A -85,B 0,C 180,E1 -11960.214,E2 -11960.214} C_VEL
LIN {X 0,Y 381.996,Z 619.812,A -85,B 0,C 180,E1 -11962.068,E2 -11962.068} C_VEL
LIN {X 0,Y 381.675,Z 624.715,A -85,B 0,C 180,E1 -11963.899,E2 -11963.899} C_VEL
LIN {X 0,Y 381.619,Z 628.3,A -85,B 0,C 180,E1 -11965.775,E2 -11965.775} C_VEL
LIN {X 0,Y 381.555,Z 630.688,A -85,B 0,C 180,E1 -11967.889,E2 -11967.889} C_VEL
LIN {X 0,Y 381.59,Z 631.297,A -85,B 0,C 180,E1 -11968.944,E2 -11968.944} C_VEL
LIN {X 0,Y 381.604,Z 631.512,A -85,B 0,C 180,E1 -11970,E2 -11970} C_VEL
LIN {X 0,Y 381.59,Z 631.294,A -85,B 0,C 180,E1 -11971.055,E2 -11971.055} C_VEL
LIN {X 0,Y 381.555,Z 630.684,A -85,B 0,C 180,E1 -11972.111,E2 -11972.111} C_VEL
LIN {X 0,Y 381.619,Z 628.291,A -85,B 0,C 180,E1 -11974.224,E2 -11974.224} C_VEL
LIN {X 0,Y 381.691,Z 624.641,A -85,B 0,C 180,E1 -11976.124,E2 -11976.124} C_VEL
LIN {X 0,Y 381.995,Z 619.786,A -85,B 0,C 180,E1 -11977.931,E2 -11977.931} C_VEL
LIN {X 0,Y 382.388,Z 614.258,A -85,B 0,C 180,E1 -11979.521,E2 -11979.521} C_VEL
LIN {X 0,Y 382.965,Z 607.357,A -85,B 0,C 180,E1 -11981.11,E2 -11981.11} C_VEL
LIN {X 0,Y 383.865,Z 598.728,A -85,B 0,C 180,E1 -11982.691,E2 -11982.691} C_VEL
LIN {X 0,Y 384.754,Z 588.809,A -85,B 0,C 180,E1 -11984.153,E2 -11984.153} C_VEL
LIN {X 0,Y 385.615,Z 578.982,A -85,B 0,C 180,E1 -11985.323,E2 -11985.323} C_VEL
LIN {X 0,Y 386.554,Z 567.987,A -85,B 0,C 180,E1 -11986.368,E2 -11986.368} C_VEL
LIN {X 0,Y 387.546,Z 555.663,A -85,B 0,C 180,E1 -11987.275,E2 -11987.275} C_VEL
LIN {X 0,Y 388.343,Z 543.993,A -85,B 0,C 180,E1 -11987.918,E2 -11987.918} C_VEL
LIN {X 0,Y 388.917,Z 531.548,A -85,B 0,C 180,E1 -11988.401,E2 -11988.401} C_VEL
LIN {X 0,Y 389.361,Z 515.677,A -85,B 0,C 180,E1 -11988.755,E2 -11988.755} C_VEL
LIN {X 0,Y 390.052,Z 447.648,A -85,B 0,C 180,E1 -11990.02,E2 -11990.02} C_VEL
LIN {X 0,Y 385.271,Z 419.09,A -85,B 0,C 180,E1 -11990.855,E2 -11990.855} C_VEL
LIN {X 0,Y 386.538,Z 404.622,A -85,B 0,C 180,E1 -11994.102,E2 -11994.102} C_VEL
LIN {X 0,Y 385.291,Z 396.966,A -85,B 0,C 180,E1 -11995.962,E2 -11995.962} C_VEL
LIN {X 0,Y 383.042,Z 386.273,A -85,B 0,C 180,E1 -11998.717,E2 -11998.717} C_VEL
LIN {X 0,Y 382.988,Z 386.275,A -85,B 0,C 180,E1 -12002.422,E2 -12002.422} C_VEL
LIN {X 0,Y 383.027,Z 386.27,A -85,B 0,C 180,E1 -12005.955,E2 -12005.955} C_VEL
LIN {X 0,Y 383.017,Z 386.272,A -85,B 0,C 180,E1 -12009.587,E2 -12009.587} C_VEL
LIN {X 0,Y 383.006,Z 386.277,A -85,B 0,C 180,E1 -12012.779,E2 -12012.779} C_VEL
LIN {X 0,Y 383.001,Z 386.273,A -85,B 0,C 180,E1 -12015.79,E2 -12015.79} C_VEL
LIN {X 0,Y 382.991,Z 386.28,A -85,B 0,C 180,E1 -12018.795,E2 -12018.795} C_VEL
LIN {X 0,Y 383.001,Z 386.273,A -85,B 0,C 180,E1 -12022.096,E2 -12022.096} C_VEL
LIN {X 0,Y 383.019,Z 386.272,A -85,B 0,C 180,E1 -12025.332,E2 -12025.332} C_VEL
LIN {X 0,Y 382.985,Z 386.278,A -85,B 0,C 180,E1 -12029.082,E2 -12029.082} C_VEL
LIN {X 0,Y 383.058,Z 386.272,A -85,B 0,C 180,E1 -12032.698,E2 -12032.698} C_VEL
LIN {X 0,Y 383.054,Z 386.269,A -85,B 0,C 180,E1 -12035.04,E2 -12035.04} C_VEL
LIN {X 0,Y 383.001,Z 386.279,A -85,B 0,C 180,E1 -12038.469,E2 -12038.469} C_VEL
LIN {X 0,Y 383.065,Z 386.266,A -85,B 0,C 180,E1 -12041.827,E2 -12041.827} C_VEL
LIN {X 0,Y 383.115,Z 386.26,A -85,B 0,C 180,E1 -12045.118,E2 -12045.118} C_VEL
LIN {X 0,Y 383.11,Z 386.266,A -85,B 0,C 180,E1 -12048.358,E2 -12048.358} C_VEL
LIN {X 0,Y 383.23,Z 386.248,A -85,B 0,C 180,E1 -12052.013,E2 -12052.013} C_VEL
LIN {X 0,Y 383.198,Z 386.25,A -85,B 0,C 180,E1 -12054.739,E2 -12054.739} C_VEL
LIN {X 0,Y 383.388,Z 386.228,A -85,B 0,C 180,E1 -12057.899,E2 -12057.899} C_VEL
LIN {X 0,Y 383.52,Z 386.213,A -85,B 0,C 180,E1 -12060,E2 -12060} C_VEL
LIN {X 0,Y 383.255,Z 386.241,A -85,B 0,C 180,E1 -12063.154,E2 -12063.154} C_VEL
LIN {X 0,Y 383.272,Z 386.241,A -85,B 0,C 180,E1 -12066.636,E2 -12066.636} C_VEL
LIN {X 0,Y 383.262,Z 386.243,A -85,B 0,C 180,E1 -12068.436,E2 -12068.436} C_VEL
LIN {X 0,Y 383.1,Z 386.263,A -85,B 0,C 180,E1 -12071.642,E2 -12071.642} C_VEL
LIN {X 0,Y 383.113,Z 386.259,A -85,B 0,C 180,E1 -12074.882,E2 -12074.882} C_VEL
LIN {X 0,Y 383.096,Z 386.265,A -85,B 0,C 180,E1 -12078.172,E2 -12078.172} C_VEL
LIN {X 0,Y 383.007,Z 386.275,A -85,B 0,C 180,E1 -12081.53,E2 -12081.53} C_VEL
LIN {X 0,Y 383.054,Z 386.266,A -85,B 0,C 180,E1 -12084.96,E2 -12084.96} C_VEL
LIN {X 0,Y 383.051,Z 386.267,A -85,B 0,C 180,E1 -12088.492,E2 -12088.492} C_VEL
LIN {X 0,Y 383.013,Z 386.274,A -85,B 0,C 180,E1 -12092.15,E2 -12092.15} C_VEL
LIN {X 0,Y 383.02,Z 386.271,A -85,B 0,C 180,E1 -12094.668,E2 -12094.668} C_VEL
LIN {X 0,Y 383.004,Z 386.276,A -85,B 0,C 180,E1 -12097.904,E2 -12097.904} C_VEL
LIN {X 0,Y 383,Z 386.277,A -85,B 0,C 180,E1 -12101.346,E2 -12101.346} C_VEL
LIN {X 0,Y 383,Z 386.273,A -85,B 0,C 180,E1 -12104.304,E2 -12104.304} C_VEL
LIN {X 0,Y 383.012,Z 386.276,A -85,B 0,C 180,E1 -12107.24,E2 -12107.24} C_VEL
LIN {X 0,Y 383.017,Z 386.271,A -85,B 0,C 180,E1 -12110.414,E2 -12110.414} C_VEL
LIN {X 0,Y 383.029,Z 386.27,A -85,B 0,C 180,E1 -12114.045,E2 -12114.045} C_VEL
LIN {X 0,Y 382.989,Z 386.278,A -85,B 0,C 180,E1 -12117.578,E2 -12117.578} C_VEL
LIN {X 0,Y 382.994,Z 386.274,A -85,B 0,C 180,E1 -12120.3,E2 -12120.3} C_VEL
LIN {X 0,Y 383.059,Z 386.267,A -85,B 0,C 180,E1 -12122.698,E2 -12122.698} C_VEL
LIN {X 0,Y 383.116,Z 386.399,A -85,B 0,C 180,E1 -12124.754,E2 -12124.754} C_VEL
LIN {X 0,Y 385.381,Z 398.071,A -85,B 0,C 180,E1 -12128.001,E2 -12128.001} C_VEL
LIN {X 0,Y 385.614,Z 402.842,A -85,B 0,C 180,E1 -12129.241,E2 -12129.241} C_VEL
LIN {X 0,Y 390.457,Z 426.83,A -85,B 0,C 180,E1 -12129.979,E2 -12129.979} C_VEL
LIN {X 0,Y 389.296,Z 510.383,A -85,B 0,C 180,E1 -12131.549,E2 -12131.549} C_VEL
LIN {X 0,Y 388.681,Z 524.195,A -85,B 0,C 180,E1 -12132.03,E2 -12132.03} C_VEL
LIN {X 0,Y 388.006,Z 536.569,A -85,B 0,C 180,E1 -12132.679,E2 -12132.679} C_VEL
LIN {X 0,Y 387.206,Z 548.408,A -85,B 0,C 180,E1 -12133.525,E2 -12133.525} C_VEL
LIN {X 0,Y 386.287,Z 560.429,A -85,B 0,C 180,E1 -12134.638,E2 -12134.638} C_VEL
LIN {X 0,Y 385.482,Z 570.003,A -85,B 0,C 180,E1 -12135.752,E2 -12135.752} C_VEL
LIN {X 0,Y 384.567,Z 579.189,A -85,B 0,C 180,E1 -12137.064,E2 -12137.064} C_VEL
LIN {X 0,Y 383.66,Z 588.109,A -85,B 0,C 180,E1 -12138.643,E2 -12138.643} C_VEL
LIN {X 0,Y 382.956,Z 595.289,A -85,B 0,C 180,E1 -12140.227,E2 -12140.227} C_VEL
LIN {X 0,Y 382.472,Z 600.132,A -85,B 0,C 180,E1 -12141.547,E2 -12141.547} C_VEL
LIN {X 0,Y 382.082,Z 605.417,A -85,B 0,C 180,E1 -12143.353,E2 -12143.353} C_VEL
LIN {X 0,Y 381.913,Z 608.437,A -85,B 0,C 180,E1 -12144.721,E2 -12144.721} C_VEL
LIN {X 0,Y 381.726,Z 610.299,A -85,B 0,C 180,E1 -12145.777,E2 -12145.777} C_VEL
LIN {X 0,Y 381.647,Z 611.7,A -85,B 0,C 180,E1 -12146.833,E2 -12146.833} C_VEL
LIN {X 0,Y 381.643,Z 612.695,A -85,B 0,C 180,E1 -12147.889,E2 -12147.889} C_VEL
LIN {X 0,Y 381.626,Z 613.309,A -85,B 0,C 180,E1 -12148.945,E2 -12148.945} C_VEL
LIN {X 0,Y 381.606,Z 613.542,A -85,B 0,C 180,E1 -12150,E2 -12150} C_VEL
LIN {X 0,Y 381.626,Z 613.352,A -85,B 0,C 180,E1 -12151.055,E2 -12151.055} C_VEL
LIN {X 0,Y 381.643,Z 612.767,A -85,B 0,C 180,E1 -12152.111,E2 -12152.111} C_VEL
LIN {X 0,Y 381.722,Z 610.444,A -85,B 0,C 180,E1 -12154.224,E2 -12154.224} C_VEL
LIN {X 0,Y 381.977,Z 607.573,A -85,B 0,C 180,E1 -12155.808,E2 -12155.808} C_VEL
LIN {X 0,Y 382.208,Z 603.685,A -85,B 0,C 180,E1 -12157.396,E2 -12157.396} C_VEL
LIN {X 0,Y 382.622,Z 598.666,A -85,B 0,C 180,E1 -12158.982,E2 -12158.982} C_VEL
LIN {X 0,Y 383.227,Z 592.348,A -85,B 0,C 180,E1 -12160.568,E2 -12160.568} C_VEL
LIN {X 0,Y 384.04,Z 583.938,A -85,B 0,C 180,E1 -12162.24,E2 -12162.24} C_VEL
LIN {X 0,Y 383.79,Z 580.131,A -85,B 0,C 180,E1 -12162.912,E2 -12162.912} C_VEL
LIN {X 0,Y 381.623,Z 573.689,A -85,B 0,C 180,E1 -12163.994,E2 -12163.994} C_VEL
LIN {X 0,Y 379.486,Z 566.779,A -85,B 0,C 180,E1 -12165.015,E2 -12165.015} C_VEL
LIN {X 0,Y 379.278,Z 562.146,A -85,B 0,C 180,E1 -12165.58,E2 -12165.58} C_VEL
LIN {X 0,Y 380.205,Z 551.303,A -85,B 0,C 180,E1 -12166.65,E2 -12166.65} C_VEL
LIN {X 0,Y 381.119,Z 539.189,A -85,B 0,C 180,E1 -12167.576,E2 -12167.576} C_VEL
LIN {X 0,Y 381.919,Z 526.497,A -85,B 0,C 180,E1 -12168.3,E2 -12168.3} C_VEL
LIN {X 0,Y 382.493,Z 513.869,A -85,B 0,C 180,E1 -12168.792,E2 -12168.792} C_VEL
LIN {X 0,Y 382.855,Z 499.528,A -85,B 0,C 180,E1 -12169.121,E2 -12169.121} C_VEL
LIN {X 0,Y 383.702,Z 427.23,A -85,B 0,C 180,E1 -12170.487,E2 -12170.487} C_VEL
LIN {X 0,Y 378.785,Z 402.96,A -85,B 0,C 180,E1 -12171.263,E2 -12171.263} C_VEL
LIN {X 0,Y 378.111,Z 397.829,A -85,B 0,C 180,E1 -12172.658,E2 -12172.658} C_VEL
LIN {X 0,Y 376.053,Z 387.148,A -85,B 0,C 180,E1 -12175.748,E2 -12175.748} C_VEL
LIN {X 0,Y 375.974,Z 387.152,A -85,B 0,C 180,E1 -12179.079,E2 -12179.079} C_VEL
LIN {X 0,Y 375.952,Z 387.157,A -85,B 0,C 180,E1 -12182.829,E2 -12182.829} C_VEL
LIN {X 0,Y 375.961,Z 387.151,A -85,B 0,C 180,E1 -12185.416,E2 -12185.416} C_VEL
LIN {X 0,Y 375.977,Z 387.15,A -85,B 0,C 180,E1 -12188.271,E2 -12188.271} C_VEL
LIN {X 0,Y 375.938,Z 387.153,A -85,B 0,C 180,E1 -12191.601,E2 -12191.601} C_VEL
LIN {X 0,Y 375.932,Z 387.154,A -85,B 0,C 180,E1 -12195.268,E2 -12195.268} C_VEL
LIN {X 0,Y 375.949,Z 387.157,A -85,B 0,C 180,E1 -12198.397,E2 -12198.397} C_VEL
LIN {X 0,Y 375.98,Z 387.148,A -85,B 0,C 180,E1 -12201.729,E2 -12201.729} C_VEL
LIN {X 0,Y 375.984,Z 387.147,A -85,B 0,C 180,E1 -12205.333,E2 -12205.333} C_VEL
LIN {X 0,Y 375.964,Z 387.155,A -85,B 0,C 180,E1 -12208.438,E2 -12208.438} C_VEL
LIN {X 0,Y 376.007,Z 387.149,A -85,B 0,C 180,E1 -12212.142,E2 -12212.142} C_VEL
LIN {X 0,Y 376.011,Z 387.147,A -85,B 0,C 180,E1 -12214.539,E2 -12214.539} C_VEL
LIN {X 0,Y 375.976,Z 387.153,A -85,B 0,C 180,E1 -12218.046,E2 -12218.046} C_VEL
LIN {X 0,Y 376.035,Z 387.142,A -85,B 0,C 180,E1 -12221.474,E2 -12221.474} C_VEL
LIN {X 0,Y 376.063,Z 387.138,A -85,B 0,C 180,E1 -12224.833,E2 -12224.833} C_VEL
LIN {X 0,Y 376.055,Z 387.144,A -85,B 0,C 180,E1 -12228.137,E2 -12228.137} C_VEL
LIN {X 0,Y 376.263,Z 387.118,A -85,B 0,C 180,E1 -12231.877,E2 -12231.877} C_VEL
LIN {X 0,Y 376.177,Z 387.124,A -85,B 0,C 180,E1 -12234.64,E2 -12234.64} C_VEL
LIN {X 0,Y 376.357,Z 387.107,A -85,B 0,C 180,E1 -12237.86,E2 -12237.86} C_VEL
LIN {X 0,Y 376.492,Z 387.089,A -85,B 0,C 180,E1 -12240,E2 -12240} C_VEL
LIN {X 0,Y 376.191,Z 387.123,A -85,B 0,C 180,E1 -12243.213,E2 -12243.213} C_VEL
LIN {X 0,Y 376.237,Z 387.116,A -85,B 0,C 180,E1 -12246.435,E2 -12246.435} C_VEL
LIN {X 0,Y 376.122,Z 387.137,A -85,B 0,C 180,E1 -12249.681,E2 -12249.681} C_VEL
LIN {X 0,Y 376.094,Z 387.14,A -85,B 0,C 180,E1 -12253.658,E2 -12253.658} C_VEL
LIN {X 0,Y 376.048,Z 387.145,A -85,B 0,C 180,E1 -12257.607,E2 -12257.607} C_VEL
LIN {X 0,Y 375.982,Z 387.148,A -85,B 0,C 180,E1 -12260.832,E2 -12260.832} C_VEL
LIN {X 0,Y 375.998,Z 387.146,A -85,B 0,C 180,E1 -12264.281,E2 -12264.281} C_VEL
LIN {X 0,Y 376.024,Z 387.143,A -85,B 0,C 180,E1 -12266.652,E2 -12266.652} C_VEL
LIN {X 0,Y 375.968,Z 387.149,A -85,B 0,C 180,E1 -12270.312,E2 -12270.312} C_VEL
LIN {X 0,Y 375.963,Z 387.15,A -85,B 0,C 180,E1 -12274.111,E2 -12274.111} C_VEL
LIN {X 0,Y 375.956,Z 387.152,A -85,B 0,C 180,E1 -12276.741,E2 -12276.741} C_VEL
LIN {X 0,Y 375.991,Z 387.146,A -85,B 0,C 180,E1 -12279.97,E2 -12279.97} C_VEL
LIN {X 0,Y 375.934,Z 387.154,A -85,B 0,C 180,E1 -12283.765,E2 -12283.765} C_VEL
LIN {X 0,Y 375.937,Z 387.157,A -85,B 0,C 180,E1 -12286.81,E2 -12286.81} C_VEL
LIN {X 0,Y 375.966,Z 387.151,A -85,B 0,C 180,E1 -12290.537,E2 -12290.537} C_VEL
LIN {X 0,Y 375.967,Z 387.151,A -85,B 0,C 180,E1 -12293.495,E2 -12293.495} C_VEL
LIN {X 0,Y 375.963,Z 387.15,A -85,B 0,C 180,E1 -12295.888,E2 -12295.888} C_VEL
LIN {X 0,Y 375.968,Z 387.154,A -85,B 0,C 180,E1 -12299.687,E2 -12299.687} C_VEL
LIN {X 0,Y 376.001,Z 387.219,A -85,B 0,C 180,E1 -12300.998,E2 -12300.998} C_VEL
LIN {X 0,Y 378.29,Z 398.1,A -85,B 0,C 180,E1 -12303.817,E2 -12303.817} C_VEL
LIN {X 0,Y 379.603,Z 405.174,A -85,B 0,C 180,E1 -12305.583,E2 -12305.583} C_VEL
LIN {X 0,Y 378.81,Z 414.414,A -85,B 0,C 180,E1 -12307.703,E2 -12307.703} C_VEL
LIN {X 0,Y 378.425,Z 419.013,A -85,B 0,C 180,E1 -12308.756,E2 -12308.756} C_VEL
LIN {X 0,Y 383.184,Z 447.025,A -85,B 0,C 180,E1 -12309.586,E2 -12309.586} C_VEL
LIN {X 0,Y 383.568,Z 451.786,A -85,B 0,C 180,E1 -12309.7,E2 -12309.7} C_VEL
LIN {X 0,Y 382.41,Z 527.154,A -85,B 0,C 180,E1 -12311.135,E2 -12311.135} C_VEL
LIN {X 0,Y 381.844,Z 539.616,A -85,B 0,C 180,E1 -12311.558,E2 -12311.558} C_VEL
LIN {X 0,Y 380.958,Z 552.513,A -85,B 0,C 180,E1 -12312.208,E2 -12312.208} C_VEL
LIN {X 0,Y 380.024,Z 564.761,A -85,B 0,C 180,E1 -12313.065,E2 -12313.065} C_VEL
LIN {X 0,Y 378.972,Z 576.344,A -85,B 0,C 180,E1 -12314.125,E2 -12314.125} C_VEL
LIN {X 0,Y 377.996,Z 587.132,A -85,B 0,C 180,E1 -12315.371,E2 -12315.371} C_VEL
LIN {X 0,Y 377.097,Z 596.983,A -85,B 0,C 180,E1 -12316.802,E2 -12316.802} C_VEL
LIN {X 0,Y 376.121,Z 605.911,A -85,B 0,C 180,E1 -12318.412,E2 -12318.412} C_VEL
LIN {X 0,Y 375.439,Z 613.098,A -85,B 0,C 180,E1 -12320.028,E2 -12320.028} C_VEL
LIN {X 0,Y 375.062,Z 617.951,A -85,B 0,C 180,E1 -12321.378,E2 -12321.378} C_VEL
LIN {X 0,Y 374.727,Z 622.668,A -85,B 0,C 180,E1 -12322.998,E2 -12322.998} C_VEL
LIN {X 0,Y 374.559,Z 626.273,A -85,B 0,C 180,E1 -12324.617,E2 -12324.617} C_VEL
LIN {X 0,Y 374.525,Z 628.133,A -85,B 0,C 180,E1 -12325.695,E2 -12325.695} C_VEL
LIN {X 0,Y 374.453,Z 630.521,A -85,B 0,C 180,E1 -12327.849,E2 -12327.849} C_VEL
LIN {X 0,Y 374.49,Z 631.13,A -85,B 0,C 180,E1 -12328.924,E2 -12328.924} C_VEL
LIN {X 0,Y 374.506,Z 631.345,A -85,B 0,C 180,E1 -12330,E2 -12330} C_VEL
LIN {X 0,Y 374.489,Z 631.126,A -85,B 0,C 180,E1 -12331.075,E2 -12331.075} C_VEL
LIN {X 0,Y 374.453,Z 629.52,A -85,B 0,C 180,E1 -12333.228,E2 -12333.228} C_VEL
LIN {X 0,Y 374.525,Z 628.123,A -85,B 0,C 180,E1 -12334.305,E2 -12334.305} C_VEL
LIN {X 0,Y 374.587,Z 624.862,A -85,B 0,C 180,E1 -12336.072,E2 -12336.072} C_VEL
LIN {X 0,Y 374.929,Z 619.617,A -85,B 0,C 180,E1 -12338.082,E2 -12338.082} C_VEL
LIN {X 0,Y 375.36,Z 614.088,A -85,B 0,C 180,E1 -12339.701,E2 -12339.701} C_VEL
LIN {X 0,Y 375.97,Z 607.188,A -85,B 0,C 180,E1 -12341.319,E2 -12341.319} C_VEL
LIN {X 0,Y 376.925,Z 598.558,A -85,B 0,C 180,E1 -12342.929,E2 -12342.929} C_VEL
LIN {X 0,Y 377.809,Z 589.037,A -85,B 0,C 180,E1 -12344.363,E2 -12344.363} C_VEL
LIN {X 0,Y 378.751,Z 578.811,A -85,B 0,C 180,E1 -12345.608,E2 -12345.608} C_VEL
LIN {X 0,Y 379.743,Z 567.816,A -85,B 0,C 180,E1 -12346.67,E2 -12346.67} C_VEL
LIN {X 0,Y 380.781,Z 555.49,A -85,B 0,C 180,E1 -12347.591,E2 -12347.591} C_VEL
LIN {X 0,Y 381.607,Z 543.819,A -85,B 0,C 180,E1 -12348.245,E2 -12348.245} C_VEL
LIN {X 0,Y 382.173,Z 531.368,A -85,B 0,C 180,E1 -12348.738,E2 -12348.738} C_VEL
LIN {X 0,Y 382.664,Z 515.49,A -85,B 0,C 180,E1 -12349.095,E2 -12349.095} C_VEL
LIN {X 0,Y 383.389,Z 448.416,A -85,B 0,C 180,E1 -12350.364,E2 -12350.364} C_VEL
LIN {X 0,Y 378.394,Z 418.991,A -85,B 0,C 180,E1 -12351.236,E2 -12351.236} C_VEL
LIN {X 0,Y 379.583,Z 406.736,A -85,B 0,C 180,E1 -12354.037,E2 -12354.037} C_VEL
LIN {X 0,Y 378.817,Z 400.531,A -85,B 0,C 180,E1 -12355.553,E2 -12355.553} C_VEL
LIN {X 0,Y 376.326,Z 388.568,A -85,B 0,C 180,E1 -12358.629,E2 -12358.629} C_VEL
LIN {X 0,Y 375.993,Z 387.152,A -85,B 0,C 180,E1 -12359.039,E2 -12359.039} C_VEL
LIN {X 0,Y 375.95,Z 387.155,A -85,B 0,C 180,E1 -12362.828,E2 -12362.828} C_VEL
LIN {X 0,Y 375.959,Z 387.153,A -85,B 0,C 180,E1 -12365.415,E2 -12365.415} C_VEL
LIN {X 0,Y 375.976,Z 387.149,A -85,B 0,C 180,E1 -12368.27,E2 -12368.27} C_VEL
LIN {X 0,Y 375.936,Z 387.154,A -85,B 0,C 180,E1 -12371.601,E2 -12371.601} C_VEL
LIN {X 0,Y 375.956,Z 387.153,A -85,B 0,C 180,E1 -12375.264,E2 -12375.264} C_VEL
LIN {X 0,Y 375.943,Z 387.156,A -85,B 0,C 180,E1 -12379.133,E2 -12379.133} C_VEL
LIN {X 0,Y 375.966,Z 387.149,A -85,B 0,C 180,E1 -12381.912,E2 -12381.912} C_VEL
LIN {X 0,Y 375.981,Z 387.149,A -85,B 0,C 180,E1 -12385.333,E2 -12385.333} C_VEL
LIN {X 0,Y 375.959,Z 387.154,A -85,B 0,C 180,E1 -12388.438,E2 -12388.438} C_VEL
LIN {X 0,Y 375.985,Z 387.149,A -85,B 0,C 180,E1 -12392.14,E2 -12392.14} C_VEL
LIN {X 0,Y 376.008,Z 387.15,A -85,B 0,C 180,E1 -12394.539,E2 -12394.539} C_VEL
LIN {X 0,Y 375.97,Z 387.151,A -85,B 0,C 180,E1 -12398.046,E2 -12398.046} C_VEL
LIN {X 0,Y 376.011,Z 387.144,A -85,B 0,C 180,E1 -12401.473,E2 -12401.473} C_VEL
LIN {X 0,Y 376.062,Z 387.14,A -85,B 0,C 180,E1 -12404.833,E2 -12404.833} C_VEL
LIN {X 0,Y 376.061,Z 387.141,A -85,B 0,C 180,E1 -12408.137,E2 -12408.137} C_VEL
LIN {X 0,Y 376.202,Z 387.122,A -85,B 0,C 180,E1 -12411.939,E2 -12411.939} C_VEL
LIN {X 0,Y 376.17,Z 387.127,A -85,B 0,C 180,E1 -12414.64,E2 -12414.64} C_VEL
LIN {X 0,Y 376.354,Z 387.104,A -85,B 0,C 180,E1 -12417.86,E2 -12417.86} C_VEL
LIN {X 0,Y 376.49,Z 387.088,A -85,B 0,C 180,E1 -12420,E2 -12420} C_VEL
LIN {X 0,Y 376.193,Z 387.121,A -85,B 0,C 180,E1 -12423.213,E2 -12423.213} C_VEL
LIN {X 0,Y 376.237,Z 387.117,A -85,B 0,C 180,E1 -12426.627,E2 -12426.627} C_VEL
LIN {X 0,Y 376.207,Z 387.121,A -85,B 0,C 180,E1 -12428.595,E2 -12428.595} C_VEL
LIN {X 0,Y 376.052,Z 387.143,A -85,B 0,C 180,E1 -12431.863,E2 -12431.863} C_VEL
LIN {X 0,Y 376.061,Z 387.138,A -85,B 0,C 180,E1 -12435.167,E2 -12435.167} C_VEL
LIN {X 0,Y 376.032,Z 387.142,A -85,B 0,C 180,E1 -12438.526,E2 -12438.526} C_VEL
LIN {X 0,Y 375.974,Z 387.154,A -85,B 0,C 180,E1 -12441.954,E2 -12441.954} C_VEL
LIN {X 0,Y 376.009,Z 387.147,A -85,B 0,C 180,E1 -12445.461,E2 -12445.461} C_VEL
LIN {X 0,Y 375.978,Z 387.148,A -85,B 0,C 180,E1 -12449.079,E2 -12449.079} C_VEL
LIN {X 0,Y 375.953,Z 387.151,A -85,B 0,C 180,E1 -12452.828,E2 -12452.828} C_VEL
LIN {X 0,Y 375.96,Z 387.154,A -85,B 0,C 180,E1 -12455.415,E2 -12455.415} C_VEL
LIN {X 0,Y 375.978,Z 387.149,A -85,B 0,C 180,E1 -12458.271,E2 -12458.271} C_VEL
LIN {X 0,Y 375.947,Z 387.158,A -85,B 0,C 180,E1 -12461.603,E2 -12461.603} C_VEL
LIN {X 0,Y 375.93,Z 387.158,A -85,B 0,C 180,E1 -12465.268,E2 -12465.268} C_VEL
LIN {X 0,Y 375.936,Z 387.153,A -85,B 0,C 180,E1 -12468.399,E2 -12468.399} C_VEL
LIN {X 0,Y 375.978,Z 387.151,A -85,B 0,C 180,E1 -12471.729,E2 -12471.729} C_VEL
LIN {X 0,Y 375.982,Z 387.154,A -85,B 0,C 180,E1 -12475.333,E2 -12475.333} C_VEL
LIN {X 0,Y 375.96,Z 387.15,A -85,B 0,C 180,E1 -12478.438,E2 -12478.438} C_VEL
LIN {X 0,Y 375.998,Z 387.145,A -85,B 0,C 180,E1 -12482.142,E2 -12482.142} C_VEL
LIN {X 0,Y 376.068,Z 387.21,A -85,B 0,C 180,E1 -12484.428,E2 -12484.428} C_VEL
LIN {X 0,Y 378.224,Z 398.426,A -85,B 0,C 180,E1 -12487.61,E2 -12487.61} C_VEL
LIN {X 0,Y 378.743,Z 402.945,A -85,B 0,C 180,E1 -12488.828,E2 -12488.828} C_VEL
LIN {X 0,Y 383.688,Z 427.167,A -85,B 0,C 180,E1 -12489.613,E2 -12489.613} C_VEL
LIN {X 0,Y 383.518,Z 447.762,A -85,B 0,C 180,E1 -12490.006,E2 -12490.006} C_VEL
LIN {X 0,Y 382.578,Z 510.566,A -85,B 0,C 180,E1 -12491.213,E2 -12491.213} C_VEL
LIN {X 0,Y 381.944,Z 524.373,A -85,B 0,C 180,E1 -12491.702,E2 -12491.702} C_VEL
LIN {X 0,Y 381.257,Z 536.743,A -85,B 0,C 180,E1 -12492.362,E2 -12492.362} C_VEL
LIN {X 0,Y 380.407,Z 548.581,A -85,B 0,C 180,E1 -12493.222,E2 -12493.222} C_VEL
LIN {X 0,Y 379.489,Z 559.964,A -85,B 0,C 180,E1 -12494.288,E2 -12494.288} C_VEL
LIN {X 0,Y 378.616,Z 570.174,A -85,B 0,C 180,E1 -12495.488,E2 -12495.488} C_VEL
LIN {X 0,Y 377.63,Z 579.36,A -85,B 0,C 180,E1 -12496.822,E2 -12496.822} C_VEL
LIN {X 0,Y 376.696,Z 588.279,A -85,B 0,C 180,E1 -12498.43,E2 -12498.43} C_VEL
LIN {X 0,Y 375.96,Z 595.459,A -85,B 0,C 180,E1 -12500.043,E2 -12500.043} C_VEL
LIN {X 0,Y 375.44,Z 600.301,A -85,B 0,C 180,E1 -12501.387,E2 -12501.387} C_VEL
LIN {X 0,Y 375.038,Z 605.007,A -85,B 0,C 180,E1 -12503.004,E2 -12503.004} C_VEL
LIN {X 0,Y 374.841,Z 608.605,A -85,B 0,C 180,E1 -12504.621,E2 -12504.621} C_VEL
LIN {X 0,Y 374.66,Z 610.467,A -85,B 0,C 180,E1 -12505.697,E2 -12505.697} C_VEL
LIN {X 0,Y 374.558,Z 611.868,A -85,B 0,C 180,E1 -12506.773,E2 -12506.773} C_VEL
LIN {X 0,Y 374.545,Z 612.863,A -85,B 0,C 180,E1 -12507.849,E2 -12507.849} C_VEL
LIN {X 0,Y 374.528,Z 613.476,A -85,B 0,C 180,E1 -12508.925,E2 -12508.925} C_VEL
LIN {X 0,Y 374.508,Z 613.709,A -85,B 0,C 180,E1 -12510,E2 -12510} C_VEL
LIN {X 0,Y 374.528,Z 613.519,A -85,B 0,C 180,E1 -12511.075,E2 -12511.075} C_VEL
LIN {X 0,Y 374.545,Z 612.934,A -85,B 0,C 180,E1 -12512.151,E2 -12512.151} C_VEL
LIN {X 0,Y 374.655,Z 610.61,A -85,B 0,C 180,E1 -12514.303,E2 -12514.303} C_VEL
LIN {X 0,Y 374.914,Z 607.74,A -85,B 0,C 180,E1 -12515.918,E2 -12515.918} C_VEL
LIN {X 0,Y 375.157,Z 603.851,A -85,B 0,C 180,E1 -12517.535,E2 -12517.535} C_VEL
LIN {X 0,Y 375.608,Z 598.832,A -85,B 0,C 180,E1 -12519.152,E2 -12519.152} C_VEL
LIN {X 0,Y 376.221,Z 592.513,A -85,B 0,C 180,E1 -12520.767,E2 -12520.767} C_VEL
LIN {X 0,Y 377.065,Z 584.448,A -85,B 0,C 180,E1 -12522.406,E2 -12522.406} C_VEL
LIN {X 0,Y 378.131,Z 574.761,A -85,B 0,C 180,E1 -12523.982,E2 -12523.982} C_VEL
LIN {X 0,Y 379.105,Z 564.409,A -85,B 0,C 180,E1 -12525.321,E2 -12525.321} C_VEL
LIN {X 0,Y 379.278,Z 562.146,A -85,B 0,C 180,E1 -12525.58,E2 -12525.58} C_VEL
LIN {X 0,Y 379.064,Z 557.423,A -85,B 0,C 180,E1 -12526.12,E2 -12526.12} C_VEL
LIN {X 0,Y 376.923,Z 549.571,A -85,B 0,C 180,E1 -12526.989,E2 -12526.989} C_VEL
LIN {X 0,Y 374.819,Z 541.303,A -85,B 0,C 180,E1 -12527.755,E2 -12527.755} C_VEL
LIN {X 0,Y 374.642,Z 535.938,A -85,B 0,C 180,E1 -12528.125,E2 -12528.125} C_VEL
LIN {X 0,Y 375.406,Z 522.937,A -85,B 0,C 180,E1 -12528.806,E2 -12528.806} C_VEL
LIN {X 0,Y 375.909,Z 509.402,A -85,B 0,C 180,E1 -12529.275,E2 -12529.275} C_VEL
LIN {X 0,Y 376.861,Z 453.406,A -85,B 0,C 180,E1 -12530.356,E2 -12530.356} C_VEL
LIN {X 0,Y 377.133,Z 428.488,A -85,B 0,C 180,E1 -12530.838,E2 -12530.838} C_VEL
LIN {X 0,Y 371.973,Z 403.821,A -85,B 0,C 180,E1 -12531.644,E2 -12531.644} C_VEL
LIN {X 0,Y 371.834,Z 403.111,A -85,B 0,C 180,E1 -12531.684,E2 -12531.684} C_VEL
LIN {X 0,Y 369.885,Z 392.469,A -85,B 0,C 180,E1 -12534.709,E2 -12534.709} C_VEL
LIN {X 0,Y 368.996,Z 388.024,A -85,B 0,C 180,E1 -12536.041,E2 -12536.041} C_VEL
LIN {X 0,Y 368.965,Z 388.028,A -85,B 0,C 180,E1 -12538.812,E2 -12538.812} C_VEL
LIN {X 0,Y 368.901,Z 388.031,A -85,B 0,C 180,E1 -12542.238,E2 -12542.238} C_VEL
LIN {X 0,Y 368.932,Z 388.029,A -85,B 0,C 180,E1 -12545.002,E2 -12545.002} C_VEL
LIN {X 0,Y 368.912,Z 388.035,A -85,B 0,C 180,E1 -12548.64,E2 -12548.64} C_VEL
LIN {X 0,Y 368.884,Z 388.033,A -85,B 0,C 180,E1 -12552.01,E2 -12552.01} C_VEL
LIN {X 0,Y 368.89,Z 388.032,A -85,B 0,C 180,E1 -12555.177,E2 -12555.177} C_VEL
LIN {X 0,Y 368.895,Z 388.033,A -85,B 0,C 180,E1 -12558.179,E2 -12558.179} C_VEL
LIN {X 0,Y 368.915,Z 388.028,A -85,B 0,C 180,E1 -12561.359,E2 -12561.359} C_VEL
LIN {X 0,Y 368.941,Z 388.025,A -85,B 0,C 180,E1 -12565.147,E2 -12565.147} C_VEL
LIN {X 0,Y 368.933,Z 388.026,A -85,B 0,C 180,E1 -12569.047,E2 -12569.047} C_VEL
LIN {X 0,Y 368.991,Z 388.019,A -85,B 0,C 180,E1 -12571.565,E2 -12571.565} C_VEL
LIN {X 0,Y 368.962,Z 388.022,A -85,B 0,C 180,E1 -12575.225,E2 -12575.225} C_VEL
LIN {X 0,Y 368.975,Z 388.021,A -85,B 0,C 180,E1 -12578.96,E2 -12578.96} C_VEL
LIN {X 0,Y 368.997,Z 388.023,A -85,B 0,C 180,E1 -12582.257,E2 -12582.257} C_VEL
LIN {X 0,Y 369.042,Z 388.017,A -85,B 0,C 180,E1 -12586.228,E2 -12586.228} C_VEL
LIN {X 0,Y 369.072,Z 388.013,A -85,B 0,C 180,E1 -12590.132,E2 -12590.132} C_VEL
LIN {X 0,Y 369.193,Z 387.996,A -85,B 0,C 180,E1 -12592.342,E2 -12592.342} C_VEL
LIN {X 0,Y 369.15,Z 387.999,A -85,B 0,C 180,E1 -12594.538,E2 -12594.538} C_VEL
LIN {X 0,Y 369.322,Z 387.983,A -85,B 0,C 180,E1 -12597.819,E2 -12597.819} C_VEL
LIN {X 0,Y 369.462,Z 387.964,A -85,B 0,C 180,E1 -12600,E2 -12600} C_VEL
LIN {X 0,Y 369.322,Z 387.98,A -85,B 0,C 180,E1 -12602.181,E2 -12602.181} C_VEL
LIN {X 0,Y 369.196,Z 387.993,A -85,B 0,C 180,E1 -12606.558,E2 -12606.558} C_VEL
LIN {X 0,Y 369.072,Z 388.012,A -85,B 0,C 180,E1 -12609.868,E2 -12609.868} C_VEL
LIN {X 0,Y 369.042,Z 388.017,A -85,B 0,C 180,E1 -12613.773,E2 -12613.773} C_VEL
LIN {X 0,Y 369.005,Z 388.021,A -85,B 0,C 180,E1 -12617.768,E2 -12617.768} C_VEL
LIN {X 0,Y 368.934,Z 388.029,A -85,B 0,C 180,E1 -12621.219,E2 -12621.219} C_VEL
LIN {X 0,Y 368.962,Z 388.023,A -85,B 0,C 180,E1 -12624.775,E2 -12624.775} C_VEL
LIN {X 0,Y 368.967,Z 388.026,A -85,B 0,C 180,E1 -12627.203,E2 -12627.203} C_VEL
LIN {X 0,Y 368.933,Z 388.028,A -85,B 0,C 180,E1 -12630.953,E2 -12630.953} C_VEL
LIN {X 0,Y 368.932,Z 388.029,A -85,B 0,C 180,E1 -12635.001,E2 -12635.001} C_VEL
LIN {X 0,Y 368.911,Z 388.029,A -85,B 0,C 180,E1 -12638.64,E2 -12638.64} C_VEL
LIN {X 0,Y 368.885,Z 388.032,A -85,B 0,C 180,E1 -12642.009,E2 -12642.009} C_VEL
LIN {X 0,Y 368.91,Z 388.034,A -85,B 0,C 180,E1 -12645.18,E2 -12645.18} C_VEL
LIN {X 0,Y 368.886,Z 388.031,A -85,B 0,C 180,E1 -12648.177,E2 -12648.177} C_VEL
LIN {X 0,Y 368.912,Z 388.031,A -85,B 0,C 180,E1 -12651.359,E2 -12651.359} C_VEL
LIN {X 0,Y 368.939,Z 388.029,A -85,B 0,C 180,E1 -12655.146,E2 -12655.146} C_VEL
LIN {X 0,Y 368.932,Z 388.031,A -85,B 0,C 180,E1 -12659.046,E2 -12659.046} C_VEL
LIN {X 0,Y 368.974,Z 388.15,A -85,B 0,C 180,E1 -12660.667,E2 -12660.667} C_VEL
LIN {X 0,Y 371.317,Z 399.183,A -85,B 0,C 180,E1 -12663.59,E2 -12663.59} C_VEL
LIN {X 0,Y 372.68,Z 406.629,A -85,B 0,C 180,E1 -12665.488,E2 -12665.488} C_VEL
LIN {X 0,Y 371.602,Z 419.132,A -85,B 0,C 180,E1 -12668.359,E2 -12668.359} C_VEL
LIN {X 0,Y 376.628,Z 448.488,A -85,B 0,C 180,E1 -12669.247,E2 -12669.247} C_VEL
LIN {X 0,Y 376.892,Z 453.762,A -85,B 0,C 180,E1 -12669.367,E2 -12669.367} C_VEL
LIN {X 0,Y 375.696,Z 527,A -85,B 0,C 180,E1 -12670.784,E2 -12670.784} C_VEL
LIN {X 0,Y 375.073,Z 540.22,A -85,B 0,C 180,E1 -12671.248,E2 -12671.248} C_VEL
LIN {X 0,Y 374.125,Z 553.47,A -85,B 0,C 180,E1 -12671.943,E2 -12671.943} C_VEL
LIN {X 0,Y 373.23,Z 564.598,A -85,B 0,C 180,E1 -12672.748,E2 -12672.748} C_VEL
LIN {X 0,Y 372.149,Z 576.18,A -85,B 0,C 180,E1 -12673.826,E2 -12673.826} C_VEL
LIN {X 0,Y 371.094,Z 586.967,A -85,B 0,C 180,E1 -12675.093,E2 -12675.093} C_VEL
LIN {X 0,Y 370.34,Z 595.142,A -85,B 0,C 180,E1 -12676.277,E2 -12676.277} C_VEL
LIN {X 0,Y 369.479,Z 603.01,A -85,B 0,C 180,E1 -12677.643,E2 -12677.643} C_VEL
LIN {X 0,Y 368.657,Z 610.696,A -85,B 0,C 180,E1 -12679.288,E2 -12679.288} C_VEL
LIN {X 0,Y 368.019,Z 617.785,A -85,B 0,C 180,E1 -12681.212,E2 -12681.212} C_VEL
LIN {X 0,Y 367.667,Z 622.502,A -85,B 0,C 180,E1 -12682.862,E2 -12682.862} C_VEL
LIN {X 0,Y 367.47,Z 626.106,A -85,B 0,C 180,E1 -12684.512,E2 -12684.512} C_VEL
LIN {X 0,Y 367.434,Z 627.966,A -85,B 0,C 180,E1 -12685.612,E2 -12685.612} C_VEL
LIN {X 0,Y 367.37,Z 629.359,A -85,B 0,C 180,E1 -12686.71,E2 -12686.71} C_VEL
LIN {X 0,Y 367.389,Z 630.963,A -85,B 0,C 180,E1 -12688.904,E2 -12688.904} C_VEL
LIN {X 0,Y 367.409,Z 631.178,A -85,B 0,C 180,E1 -12690,E2 -12690} C_VEL
LIN {X 0,Y 367.389,Z 630.959,A -85,B 0,C 180,E1 -12691.096,E2 -12691.096} C_VEL
LIN {X 0,Y 367.37,Z 629.353,A -85,B 0,C 180,E1 -12693.29,E2 -12693.29} C_VEL
LIN {X 0,Y 367.434,Z 627.955,A -85,B 0,C 180,E1 -12694.388,E2 -12694.388} C_VEL
LIN {X 0,Y 367.484,Z 625.051,A -85,B 0,C 180,E1 -12696.02,E2 -12696.02} C_VEL
LIN {X 0,Y 367.751,Z 621.042,A -85,B 0,C 180,E1 -12697.688,E2 -12697.688} C_VEL
LIN {X 0,Y 368.222,Z 614.93,A -85,B 0,C 180,E1 -12699.614,E2 -12699.614} C_VEL
LIN {X 0,Y 368.856,Z 608.255,A -85,B 0,C 180,E1 -12701.262,E2 -12701.262} C_VEL
LIN {X 0,Y 369.797,Z 599.976,A -85,B 0,C 180,E1 -12702.903,E2 -12702.903} C_VEL
LIN {X 0,Y 370.627,Z 591.485,A -85,B 0,C 180,E1 -12704.271,E2 -12704.271} C_VEL
LIN {X 0,Y 371.652,Z 580.995,A -85,B 0,C 180,E1 -12705.633,E2 -12705.633} C_VEL
LIN {X 0,Y 372.649,Z 570.617,A -85,B 0,C 180,E1 -12706.715,E2 -12706.715} C_VEL
LIN {X 0,Y 373.701,Z 559.239,A -85,B 0,C 180,E1 -12707.653,E2 -12707.653} C_VEL
LIN {X 0,Y 374.572,Z 547.548,A -85,B 0,C 180,E1 -12708.388,E2 -12708.388} C_VEL
LIN {X 0,Y 375.331,Z 534.071,A -85,B 0,C 180,E1 -12708.986,E2 -12708.986} C_VEL
LIN {X 0,Y 375.873,Z 520.673,A -85,B 0,C 180,E1 -12709.348,E2 -12709.348} C_VEL
LIN {X 0,Y 376.782,Z 449.665,A -85,B 0,C 180,E1 -12710.709,E2 -12710.709} C_VEL
LIN {X 0,Y 371.868,Z 420.717,A -85,B 0,C 180,E1 -12711.58,E2 -12711.58} C_VEL
LIN {X 0,Y 371.541,Z 418.829,A -85,B 0,C 180,E1 -12711.645,E2 -12711.645} C_VEL
LIN {X 0,Y 372.646,Z 407.808,A -85,B 0,C 180,E1 -12714.217,E2 -12714.217} C_VEL
LIN {X 0,Y 371.799,Z 401.603,A -85,B 0,C 180,E1 -12715.77,E2 -12715.77} C_VEL
LIN {X 0,Y 369.301,Z 389.676,A -85,B 0,C 180,E1 -12718.907,E2 -12718.907} C_VEL
LIN {X 0,Y 368.935,Z 388.029,A -85,B 0,C 180,E1 -12719.395,E2 -12719.395} C_VEL
LIN {X 0,Y 368.898,Z 388.036,A -85,B 0,C 180,E1 -12723.043,E2 -12723.043} C_VEL
LIN {X 0,Y 368.919,Z 388.027,A -85,B 0,C 180,E1 -12726.197,E2 -12726.197} C_VEL
LIN {X 0,Y 368.906,Z 388.035,A -85,B 0,C 180,E1 -12728.953,E2 -12728.953} C_VEL
LIN {X 0,Y 368.882,Z 388.032,A -85,B 0,C 180,E1 -12732.009,E2 -12732.009} C_VEL
LIN {X 0,Y 368.909,Z 388.032,A -85,B 0,C 180,E1 -12735.18,E2 -12735.18} C_VEL
LIN {X 0,Y 368.885,Z 388.032,A -85,B 0,C 180,E1 -12738.178,E2 -12738.178} C_VEL
LIN {X 0,Y 368.91,Z 388.03,A -85,B 0,C 180,E1 -12741.36,E2 -12741.36} C_VEL
LIN {X 0,Y 368.938,Z 388.027,A -85,B 0,C 180,E1 -12745.147,E2 -12745.147} C_VEL
LIN {X 0,Y 368.93,Z 388.029,A -85,B 0,C 180,E1 -12749.047,E2 -12749.047} C_VEL
LIN {X 0,Y 368.964,Z 388.026,A -85,B 0,C 180,E1 -12752.797,E2 -12752.797} C_VEL
LIN {X 0,Y 368.947,Z 388.026,A -85,B 0,C 180,E1 -12756.113,E2 -12756.113} C_VEL
LIN {X 0,Y 368.939,Z 388.026,A -85,B 0,C 180,E1 -12759.947,E2 -12759.947} C_VEL
LIN {X 0,Y 368.978,Z 388.02,A -85,B 0,C 180,E1 -12763.399,E2 -12763.399} C_VEL
LIN {X 0,Y 369.062,Z 388.012,A -85,B 0,C 180,E1 -12766.79,E2 -12766.79} C_VEL
LIN {X 0,Y 369.07,Z 388.012,A -85,B 0,C 180,E1 -12770.132,E2 -12770.132} C_VEL
LIN {X 0,Y 369.192,Z 387.993,A -85,B 0,C 180,E1 -12773.442,E2 -12773.442} C_VEL
LIN {X 0,Y 369.319,Z 387.98,A -85,B 0,C 180,E1 -12777.819,E2 -12777.819} C_VEL
LIN {X 0,Y 369.459,Z 387.964,A -85,B 0,C 180,E1 -12780,E2 -12780} C_VEL
LIN {X 0,Y 369.322,Z 387.984,A -85,B 0,C 180,E1 -12782.181,E2 -12782.181} C_VEL
LIN {X 0,Y 369.207,Z 387.993,A -85,B 0,C 180,E1 -12786.615,E2 -12786.615} C_VEL
LIN {X 0,Y 369.14,Z 388,A -85,B 0,C 180,E1 -12788.761,E2 -12788.761} C_VEL
LIN {X 0,Y 369.008,Z 388.022,A -85,B 0,C 180,E1 -12792.093,E2 -12792.093} C_VEL
LIN {X 0,Y 369,Z 388.019,A -85,B 0,C 180,E1 -12795.465,E2 -12795.465} C_VEL
LIN {X 0,Y 368.992,Z 388.018,A -85,B 0,C 180,E1 -12798.892,E2 -12798.892} C_VEL
LIN {X 0,Y 368.94,Z 388.026,A -85,B 0,C 180,E1 -12802.395,E2 -12802.395} C_VEL
LIN {X 0,Y 369.002,Z 388.021,A -85,B 0,C 180,E1 -12805.98,E2 -12805.98} C_VEL
LIN {X 0,Y 368.969,Z 388.021,A -85,B 0,C 180,E1 -12808.813,E2 -12808.813} C_VEL
LIN {X 0,Y 368.902,Z 388.031,A -85,B 0,C 180,E1 -12812.238,E2 -12812.238} C_VEL
LIN {X 0,Y 368.931,Z 388.026,A -85,B 0,C 180,E1 -12815.002,E2 -12815.002} C_VEL
LIN {X 0,Y 368.913,Z 388.028,A -85,B 0,C 180,E1 -12818.641,E2 -12818.641} C_VEL
LIN {X 0,Y 368.89,Z 388.033,A -85,B 0,C 180,E1 -12822.011,E2 -12822.011} C_VEL
LIN {X 0,Y 368.883,Z 388.035,A -85,B 0,C 180,E1 -12825.176,E2 -12825.176} C_VEL
LIN {X 0,Y 368.884,Z 388.032,A -85,B 0,C 180,E1 -12828.178,E2 -12828.178} C_VEL
LIN {X 0,Y 368.912,Z 388.034,A -85,B 0,C 180,E1 -12831.359,E2 -12831.359} C_VEL
LIN {X 0,Y 368.939,Z 388.029,A -85,B 0,C 180,E1 -12835.147,E2 -12835.147} C_VEL
LIN {X 0,Y 368.931,Z 388.03,A -85,B 0,C 180,E1 -12839.047,E2 -12839.047} C_VEL
LIN {X 0,Y 368.982,Z 388.023,A -85,B 0,C 180,E1 -12841.564,E2 -12841.564} C_VEL
LIN {X 0,Y 368.998,Z 388.055,A -85,B 0,C 180,E1 -12844.096,E2 -12844.096} C_VEL
LIN {X 0,Y 371.048,Z 398.592,A -85,B 0,C 180,E1 -12847.152,E2 -12847.152} C_VEL
LIN {X 0,Y 371.772,Z 403.15,A -85,B 0,C 180,E1 -12848.422,E2 -12848.422} C_VEL
LIN {X 0,Y 375.571,Z 420.444,A -85,B 0,C 180,E1 -12849.012,E2 -12849.012} C_VEL
LIN {X 0,Y 377.197,Z 429.454,A -85,B 0,C 180,E1 -12849.288,E2 -12849.288} C_VEL
LIN {X 0,Y 375.93,Z 509.575,A -85,B 0,C 180,E1 -12850.833,E2 -12850.833} C_VEL
LIN {X 0,Y 375.323,Z 523.029,A -85,B 0,C 180,E1 -12851.297,E2 -12851.297} C_VEL
LIN {X 0,Y 374.594,Z 535.816,A -85,B 0,C 180,E1 -12851.967,E2 -12851.967} C_VEL
LIN {X 0,Y 373.745,Z 547.167,A -85,B 0,C 180,E1 -12852.773,E2 -12852.773} C_VEL
LIN {X 0,Y 372.817,Z 558.367,A -85,B 0,C 180,E1 -12853.806,E2 -12853.806} C_VEL
LIN {X 0,Y 371.863,Z 569.285,A -85,B 0,C 180,E1 -12855.078,E2 -12855.078} C_VEL
LIN {X 0,Y 370.939,Z 577.834,A -85,B 0,C 180,E1 -12856.301,E2 -12856.301} C_VEL
LIN {X 0,Y 370.034,Z 585.71,A -85,B 0,C 180,E1 -12857.663,E2 -12857.663} C_VEL
LIN {X 0,Y 369.181,Z 593.407,A -85,B 0,C 180,E1 -12859.304,E2 -12859.304} C_VEL
LIN {X 0,Y 368.406,Z 600.471,A -85,B 0,C 180,E1 -12861.222,E2 -12861.222} C_VEL
LIN {X 0,Y 367.984,Z 605.176,A -85,B 0,C 180,E1 -12862.87,E2 -12862.87} C_VEL
LIN {X 0,Y 367.773,Z 608.773,A -85,B 0,C 180,E1 -12864.517,E2 -12864.517} C_VEL
LIN {X 0,Y 367.595,Z 610.634,A -85,B 0,C 180,E1 -12865.614,E2 -12865.614} C_VEL
LIN {X 0,Y 367.473,Z 612.035,A -85,B 0,C 180,E1 -12866.711,E2 -12866.711} C_VEL
LIN {X 0,Y 367.43,Z 613.643,A -85,B 0,C 180,E1 -12868.904,E2 -12868.904} C_VEL
LIN {X 0,Y 367.411,Z 613.876,A -85,B 0,C 180,E1 -12870,E2 -12870} C_VEL
LIN {X 0,Y 367.43,Z 613.686,A -85,B 0,C 180,E1 -12871.096,E2 -12871.096} C_VEL
LIN {X 0,Y 367.471,Z 612.134,A -85,B 0,C 180,E1 -12873.289,E2 -12873.289} C_VEL
LIN {X 0,Y 367.59,Z 610.776,A -85,B 0,C 180,E1 -12874.386,E2 -12874.386} C_VEL
LIN {X 0,Y 367.842,Z 607.587,A -85,B 0,C 180,E1 -12876.191,E2 -12876.191} C_VEL
LIN {X 0,Y 368.109,Z 604.017,A -85,B 0,C 180,E1 -12877.681,E2 -12877.681} C_VEL
LIN {X 0,Y 368.578,Z 598.998,A -85,B 0,C 180,E1 -12879.328,E2 -12879.328} C_VEL
LIN {X 0,Y 369.227,Z 592.679,A -85,B 0,C 180,E1 -12880.973,E2 -12880.973} C_VEL
LIN {X 0,Y 370.121,Z 584.767,A -85,B 0,C 180,E1 -12882.613,E2 -12882.613} C_VEL
LIN {X 0,Y 371.248,Z 574.924,A -85,B 0,C 180,E1 -12884.247,E2 -12884.247} C_VEL
LIN {X 0,Y 372.179,Z 565.435,A -85,B 0,C 180,E1 -12885.51,E2 -12885.51} C_VEL
LIN {X 0,Y 373.139,Z 554.365,A -85,B 0,C 180,E1 -12886.693,E2 -12886.693} C_VEL
LIN {X 0,Y 374.122,Z 543.167,A -85,B 0,C 180,E1 -12887.633,E2 -12887.633} C_VEL
LIN {X 0,Y 374.642,Z 535.938,A -85,B 0,C 180,E1 -12888.125,E2 -12888.125} C_VEL
LIN {X 0,Y 374.324,Z 532.29,A -85,B 0,C 180,E1 -12888.371,E2 -12888.371} C_VEL
LIN {X 0,Y 371.907,Z 526.652,A -85,B 0,C 180,E1 -12888.815,E2 -12888.815} C_VEL
